LIN {X -0.093,Y -454.744,Z 848.526,A 0.000,B 0.000,C 90.000,E1 94.645} C_DIS
LIN {X 0.070,Y -444.193,Z 848.516,A 0.000,B 0.000,C 90.000,E1 92.808} C_DIS
LIN {X -0.166,Y -434.901,Z 848.507,A 0.000,B 0.000,C 90.000,E1 91.260} C_DIS
LIN {X -0.133,Y -425.303,Z 848.498,A 0.000,B 0.000,C 90.000,E1 89.656} C_DIS
LIN {X -0.064,Y -412.236,Z 848.486,A 0.000,B 0.000,C 90.000,E1 87.478} C_DIS
LIN {X 0.014,Y -402.403,Z 848.477,A 0.000,B 0.000,C 90.000,E1 85.812} C_DIS
LIN {X -0.027,Y -390.990,Z 848.466,A 0.000,B 0.000,C 90.000,E1 83.856} C_DIS
LIN {X 0.140,Y -378.162,Z 848.453,A 0.000,B 0.000,C 90.000,E1 81.546} C_DIS
LIN {X 0.095,Y -364.044,Z 848.439,A 0.000,B 0.000,C 90.000,E1 78.926} C_DIS
LIN {X -0.197,Y -351.890,Z 848.425,A 0.000,B 0.000,C 90.000,E1 76.589} C_DIS
LIN {X -0.106,Y -341.168,Z 848.414,A 0.000,B 0.000,C 90.000,E1 74.448} C_DIS
LIN {X 0.022,Y -327.690,Z 848.398,A 0.000,B 0.000,C 90.000,E1 71.638} C_DIS
LIN {X 0.142,Y -316.044,Z 848.384,A 0.000,B 0.000,C 90.000,E1 69.082} C_DIS
LIN {X -0.007,Y -301.999,Z 848.366,A 0.000,B 0.000,C 90.000,E1 65.869} C_DIS
LIN {X 0.053,Y -289.799,Z 848.349,A 0.000,B 0.000,C 90.000,E1 62.871} C_DIS
LIN {X -0.164,Y -279.159,Z 848.334,A 0.000,B 0.000,C 90.000,E1 60.205} C_DIS
LIN {X 0.005,Y -266.373,Z 848.315,A 0.000,B 0.000,C 90.000,E1 56.707} C_DIS
LIN {X 0.138,Y -254.533,Z 848.295,A 0.000,B 0.000,C 90.000,E1 53.130} C_DIS
LIN {X -0.031,Y -244.665,Z 848.277,A 0.000,B 0.000,C 90.000,E1 49.908} C_DIS
LIN {X -0.022,Y -234.511,Z 848.257,A 0.000,B 0.000,C 90.000,E1 46.215} C_DIS
LIN {X -0.016,Y -225.100,Z 848.236,A 0.000,B 0.000,C 90.000,E1 42.447} C_DIS
LIN {X 0.071,Y -218.003,Z 848.219,A 0.000,B 0.000,C 90.000,E1 39.358} C_DIS
LIN {X 0.029,Y -209.591,Z 848.197,A 0.000,B 0.000,C 90.000,E1 35.471} C_DIS
LIN {X -0.103,Y -203.336,Z 848.180,A 0.000,B 0.000,C 90.000,E1 32.339} C_DIS
LIN {X 0.075,Y -197.686,Z 848.162,A 0.000,B 0.000,C 90.000,E1 29.077} C_DIS
LIN {X 0.000,Y -192.660,Z 848.144,A 0.000,B 0.000,C 90.000,E1 25.848} C_DIS
LIN {X -0.094,Y -188.383,Z 848.125,A 0.000,B 0.000,C 90.000,E1 22.589} C_DIS
LIN {X -0.027,Y -184.224,Z 848.102,A 0.000,B 0.000,C 90.000,E1 18.417} C_DIS
LIN {X -0.080,Y -181.186,Z 848.079,A 0.000,B 0.000,C 90.000,E1 14.245} C_DIS
LIN {X -0.003,Y -178.587,Z 848.041,A 0.000,B 0.000,C 90.000,E1 7.466} C_DIS
LIN {X -0.048,Y -179.892,Z 847.979,A 0.000,B 0.000,C 90.000,E1 356.159} C_DIS
LIN {X -0.006,Y -182.801,Z 847.950,A 0.000,B 0.000,C 90.000,E1 351.084} C_DIS
LIN {X 0.036,Y -186.260,Z 847.927,A 0.000,B 0.000,C 90.000,E1 346.881} C_DIS
LIN {X 0.040,Y -190.786,Z 847.904,A 0.000,B 0.000,C 90.000,E1 342.725} C_DIS
LIN {X -0.070,Y -196.199,Z 847.881,A 0.000,B 0.000,C 90.000,E1 338.646} C_DIS
LIN {X -0.084,Y -202.510,Z 847.859,A 0.000,B 0.000,C 90.000,E1 334.588} C_DIS
LIN {X -0.101,Y -209.563,Z 847.836,A 0.000,B 0.000,C 90.000,E1 330.589} C_DIS
LIN {X -0.029,Y -217.357,Z 847.815,A 0.000,B 0.000,C 90.000,E1 326.628} C_DIS
LIN {X 0.070,Y -224.179,Z 847.797,A 0.000,B 0.000,C 90.000,E1 323.497} C_DIS
LIN {X 0.021,Y -232.765,Z 847.778,A 0.000,B 0.000,C 90.000,E1 320.070} C_DIS
LIN {X 0.005,Y -242.205,Z 847.759,A 0.000,B 0.000,C 90.000,E1 316.701} C_DIS
LIN {X 0.077,Y -252.624,Z 847.741,A 0.000,B 0.000,C 90.000,E1 313.380} C_DIS
LIN {X -0.055,Y -264.049,Z 847.723,A 0.000,B 0.000,C 90.000,E1 310.172} C_DIS
LIN {X 0.005,Y -276.404,Z 847.706,A 0.000,B 0.000,C 90.000,E1 306.996} C_DIS
LIN {X -0.026,Y -289.989,Z 847.688,A 0.000,B 0.000,C 90.000,E1 303.913} C_DIS
LIN {X -0.143,Y -304.691,Z 847.672,A 0.000,B 0.000,C 90.000,E1 300.924} C_DIS
LIN {X -0.023,Y -317.154,Z 847.659,A 0.000,B 0.000,C 90.000,E1 298.615} C_DIS
LIN {X 0.048,Y -332.889,Z 847.645,A 0.000,B 0.000,C 90.000,E1 296.052} C_DIS
LIN {X 0.102,Y -352.276,Z 847.629,A 0.000,B 0.000,C 90.000,E1 293.259} C_DIS
LIN {X 0.065,Y -371.074,Z 847.616,A 0.000,B 0.000,C 90.000,E1 290.865} C_DIS
LIN {X -0.046,Y -394.102,Z 847.602,A 0.000,B 0.000,C 90.000,E1 288.308} C_DIS
LIN {X -0.007,Y -412.240,Z 847.591,A 0.000,B 0.000,C 90.000,E1 286.386} C_DIS
LIN {X 0.017,Y -422.316,Z 847.585,A 0.000,B 0.000,C 90.000,E1 285.315} C_DIS
LIN {X -0.164,Y -434.613,Z 847.578,A 0.000,B 0.000,C 90.000,E1 284.008} C_DIS
LIN {X -0.130,Y -444.163,Z 847.572,A 0.000,B 0.000,C 90.000,E1 282.939} C_DIS
LIN {X -0.087,Y -453.154,Z 847.566,A 0.000,B 0.000,C 90.000,E1 281.883} C_DIS
LIN {X -0.023,Y -461.566,Z 847.560,A 0.000,B 0.000,C 90.000,E1 280.838} C_DIS
LIN {X 0.149,Y -469.405,Z 847.555,A 0.000,B 0.000,C 90.000,E1 279.792} C_DIS
LIN {X 0.168,Y -474.800,Z 847.550,A 0.000,B 0.000,C 90.000,E1 279.029} C_DIS
LIN {X 0.150,Y -479.624,Z 847.546,A 0.000,B 0.000,C 90.000,E1 278.276} C_DIS
LIN {X 0.114,Y -483.720,Z 847.542,A 0.000,B 0.000,C 90.000,E1 277.530} C_DIS
LIN {X 0.175,Y -487.070,Z 847.538,A 0.000,B 0.000,C 90.000,E1 276.777} C_DIS
LIN {X -0.110,Y -488.919,Z 847.535,A 0.000,B 0.000,C 90.000,E1 276.315} C_DIS
LIN {X 0.096,Y -490.405,Z 847.532,A 0.000,B 0.000,C 90.000,E1 275.796} C_DIS
LIN {X -0.176,Y -491.554,Z 847.530,A 0.000,B 0.000,C 90.000,E1 275.334} C_DIS
LIN {X 0.006,Y -492.300,Z 847.527,A 0.000,B 0.000,C 90.000,E1 274.821} C_DIS
LIN {X 0.238,Y -492.724,Z 847.524,A 0.000,B 0.000,C 90.000,E1 274.302} C_DIS
LIN {X -0.020,Y -492.771,Z 847.521,A 0.000,B 0.000,C 90.000,E1 273.841} C_DIS
LIN {X 0.185,Y -492.421,Z 847.519,A 0.000,B 0.000,C 90.000,E1 273.326} C_DIS
LIN {X -0.074,Y -491.691,Z 847.516,A 0.000,B 0.000,C 90.000,E1 272.865} C_DIS
LIN {X 0.131,Y -490.485,Z 847.513,A 0.000,B 0.000,C 90.000,E1 272.350} C_DIS
LIN {X -0.154,Y -488.845,Z 847.510,A 0.000,B 0.000,C 90.000,E1 271.892} C_DIS
LIN {X 0.057,Y -486.738,Z 847.508,A 0.000,B 0.000,C 90.000,E1 271.375} C_DIS
LIN {X 0.241,Y -483.997,Z 847.505,A 0.000,B 0.000,C 90.000,E1 270.859} C_DIS
LIN {X -0.074,Y -480.610,Z 847.502,A 0.000,B 0.000,C 90.000,E1 270.401} C_DIS
LIN {X -0.239,Y -478.699,Z 847.501,A 0.000,B 0.000,C 90.000,E1 270.172} C_DIS
LIN {X -0.100,Y -474.155,Z 847.498,A 0.000,B 0.000,C 90.000,E1 269.656} C_DIS
LIN {X 0.101,Y -468.795,Z 847.495,A 0.000,B 0.000,C 90.000,E1 269.141} C_DIS
LIN {X 0.136,Y -462.760,Z 847.493,A 0.000,B 0.000,C 90.000,E1 268.682} C_DIS
LIN {X -0.193,Y -459.346,Z 847.492,A 0.000,B 0.000,C 90.000,E1 268.511} C_DIS
LIN {X 0.175,Y -452.338,Z 847.490,A 0.000,B 0.000,C 90.000,E1 268.108} C_DIS
LIN {X 0.168,Y -445.005,Z 847.488,A 0.000,B 0.000,C 90.000,E1 267.822} C_DIS
LIN {X -0.214,Y -437.402,Z 847.487,A 0.000,B 0.000,C 90.000,E1 267.650} C_DIS
LIN {X -0.193,Y -428.427,Z 847.486,A 0.000,B 0.000,C 90.000,E1 267.478} C_DIS
LIN {X 0.039,Y -421.444,Z 847.485,A 0.000,B 0.000,C 90.000,E1 267.364} C_DIS
LIN {X 0.194,Y -415.603,Z 847.485,A 0.000,B 0.000,C 90.000,E1 267.306} C_DIS
LIN {X 0.058,Y -181.028,Z 847.485,A 0.000,B 0.000,C 90.000,E1 267.306} C_DIS
LIN {X 0.079,Y -180.786,Z 847.471,A 0.000,B 0.000,C 90.000,E1 264.723} C_DIS
LIN {X -0.027,Y -178.883,Z 847.443,A 0.000,B 0.000,C 90.000,E1 259.690} C_DIS
LIN {X 0.049,Y -175.926,Z 847.414,A 0.000,B 0.000,C 90.000,E1 254.574} C_DIS
LIN {X -0.005,Y -175.366,Z 847.410,A 0.000,B 0.000,C 90.000,E1 253.740} C_DIS
LIN {X 0.053,Y -172.144,Z 847.386,A 0.000,B 0.000,C 90.000,E1 249.444} C_DIS
LIN {X 0.030,Y -171.608,Z 847.381,A 0.000,B 0.000,C 90.000,E1 248.592} C_DIS
LIN {X 0.019,Y -167.831,Z 847.357,A 0.000,B 0.000,C 90.000,E1 244.280} C_DIS
LIN {X 0.036,Y -166.557,Z 847.347,A 0.000,B 0.000,C 90.000,E1 242.538} C_DIS
LIN {X -0.054,Y -162.551,Z 847.323,A 0.000,B 0.000,C 90.000,E1 238.201} C_DIS
LIN {X 0.006,Y -161.229,Z 847.313,A 0.000,B 0.000,C 90.000,E1 236.421} C_DIS
LIN {X 0.041,Y -157.235,Z 847.289,A 0.000,B 0.000,C 90.000,E1 231.984} C_DIS
LIN {X 0.064,Y -155.959,Z 847.279,A 0.000,B 0.000,C 90.000,E1 230.194} C_DIS
LIN {X 0.023,Y -152.213,Z 847.254,A 0.000,B 0.000,C 90.000,E1 225.729} C_DIS
LIN {X 0.043,Y -150.457,Z 847.239,A 0.000,B 0.000,C 90.000,E1 223.014} C_DIS
LIN {X 0.069,Y -147.183,Z 847.214,A 0.000,B 0.000,C 90.000,E1 218.463} C_DIS
LIN {X 0.036,Y -145.201,Z 847.194,A 0.000,B 0.000,C 90.000,E1 214.818} C_DIS
LIN {X -0.054,Y -142.338,Z 847.163,A 0.000,B 0.000,C 90.000,E1 209.333} C_DIS
LIN {X -0.001,Y -141.727,Z 847.153,A 0.000,B 0.000,C 90.000,E1 207.462} C_DIS
LIN {X -0.019,Y -139.480,Z 847.116,A 0.000,B 0.000,C 90.000,E1 200.972} C_DIS
LIN {X -0.029,Y -138.979,Z 847.101,A 0.000,B 0.000,C 90.000,E1 198.181} C_DIS
LIN {X -0.045,Y -138.332,Z 847.054,A 0.000,B 0.000,C 90.000,E1 189.782} C_DIS
LIN {X -0.044,Y -139.429,Z 847.008,A 0.000,B 0.000,C 90.000,E1 181.375} C_DIS
LIN {X 0.009,Y -141.357,Z 846.971,A 0.000,B 0.000,C 90.000,E1 174.837} C_DIS
LIN {X -0.015,Y -142.711,Z 846.956,A 0.000,B 0.000,C 90.000,E1 172.064} C_DIS
LIN {X -0.056,Y -145.085,Z 846.930,A 0.000,B 0.000,C 90.000,E1 167.465} C_DIS
LIN {X -0.061,Y -147.710,Z 846.910,A 0.000,B 0.000,C 90.000,E1 163.795} C_DIS
LIN {X 0.023,Y -150.365,Z 846.890,A 0.000,B 0.000,C 90.000,E1 160.115} C_DIS
LIN {X 0.041,Y -153.791,Z 846.869,A 0.000,B 0.000,C 90.000,E1 156.485} C_DIS
LIN {X -0.038,Y -157.204,Z 846.849,A 0.000,B 0.000,C 90.000,E1 152.922} C_DIS
LIN {X 0.043,Y -161.366,Z 846.830,A 0.000,B 0.000,C 90.000,E1 149.331} C_DIS
LIN {X 0.054,Y -165.568,Z 846.810,A 0.000,B 0.000,C 90.000,E1 145.801} C_DIS
LIN {X -0.062,Y -170.487,Z 846.791,A 0.000,B 0.000,C 90.000,E1 142.351} C_DIS
LIN {X 0.086,Y -175.367,Z 846.772,A 0.000,B 0.000,C 90.000,E1 138.852} C_DIS
LIN {X -0.051,Y -180.991,Z 846.753,A 0.000,B 0.000,C 90.000,E1 135.486} C_DIS
LIN {X 0.074,Y -186.419,Z 846.734,A 0.000,B 0.000,C 90.000,E1 132.081} C_DIS
LIN {X -0.125,Y -191.045,Z 846.720,A 0.000,B 0.000,C 90.000,E1 129.644} C_DIS
LIN {X -0.005,Y -192.945,Z 846.714,A 0.000,B 0.000,C 90.000,E1 128.463} C_DIS
LIN {X -0.055,Y -293.674,Z 846.714,A 0.000,B 0.000,C 90.000,E1 128.463} C_DIS
LIN {X -0.103,Y -294.466,Z 846.714,A 0.000,B 0.000,C 90.000,E1 128.463} C_DIS
LIN {X 0.120,Y -300.090,Z 846.712,A 0.000,B 0.000,C 90.000,E1 128.177} C_DIS
LIN {X -0.076,Y -302.819,Z 846.711,A 0.000,B 0.000,C 90.000,E1 127.971} C_DIS
LIN {X -0.016,Y -306.570,Z 846.708,A 0.000,B 0.000,C 90.000,E1 127.443} C_DIS
LIN {X -0.001,Y -308.236,Z 846.706,A 0.000,B 0.000,C 90.000,E1 127.111} C_DIS
LIN {X -0.044,Y -309.542,Z 846.704,A 0.000,B 0.000,C 90.000,E1 126.790} C_DIS
LIN {X 0.123,Y -321.746,Z 846.683,A 0.000,B 0.000,C 90.000,E1 122.880} C_DIS
LIN {X 0.002,Y -332.292,Z 846.667,A 0.000,B 0.000,C 90.000,E1 120.050} C_DIS
LIN {X -0.030,Y -344.201,Z 846.651,A 0.000,B 0.000,C 90.000,E1 117.257} C_DIS
LIN {X -0.025,Y -357.574,Z 846.636,A 0.000,B 0.000,C 90.000,E1 114.515} C_DIS
LIN {X -0.172,Y -370.791,Z 846.623,A 0.000,B 0.000,C 90.000,E1 112.153} C_DIS
LIN {X -0.133,Y -385.354,Z 846.610,A 0.000,B 0.000,C 90.000,E1 109.812} C_DIS
LIN {X 0.009,Y -401.370,Z 846.597,A 0.000,B 0.000,C 90.000,E1 107.511} C_DIS
LIN {X -0.078,Y -418.953,Z 846.585,A 0.000,B 0.000,C 90.000,E1 105.300} C_DIS
LIN {X 0.079,Y -438.195,Z 846.573,A 0.000,B 0.000,C 90.000,E1 103.119} C_DIS
LIN {X -0.120,Y -458.364,Z 846.562,A 0.000,B 0.000,C 90.000,E1 101.130} C_DIS
LIN {X -0.212,Y -468.460,Z 846.557,A 0.000,B 0.000,C 90.000,E1 100.197} C_DIS
LIN {X -0.174,Y -470.265,Z 846.555,A 0.000,B 0.000,C 90.000,E1 99.962} C_DIS
LIN {X 0.141,Y -471.770,Z 846.554,A 0.000,B 0.000,C 90.000,E1 99.670} C_DIS
LIN {X -0.087,Y -472.896,Z 846.552,A 0.000,B 0.000,C 90.000,E1 99.443} C_DIS
LIN {X 0.097,Y -474.241,Z 846.550,A 0.000,B 0.000,C 90.000,E1 98.916} C_DIS
LIN {X 0.214,Y -474.566,Z 846.547,A 0.000,B 0.000,C 90.000,E1 98.398} C_DIS
LIN {X -0.128,Y -473.929,Z 846.544,A 0.000,B 0.000,C 90.000,E1 97.936} C_DIS
LIN {X 0.063,Y -472.229,Z 846.541,A 0.000,B 0.000,C 90.000,E1 97.409} C_DIS
LIN {X -0.138,Y -470.887,Z 846.540,A 0.000,B 0.000,C 90.000,E1 97.182} C_DIS
LIN {X -0.206,Y -454.710,Z 846.526,A 0.000,B 0.000,C 90.000,E1 94.645} C_DIS
LIN {X -0.041,Y -444.143,Z 846.516,A 0.000,B 0.000,C 90.000,E1 92.808} C_DIS
LIN {X 0.159,Y -434.848,Z 846.507,A 0.000,B 0.000,C 90.000,E1 91.203} C_DIS
LIN {X 0.184,Y -425.251,Z 846.498,A 0.000,B 0.000,C 90.000,E1 89.599} C_DIS
LIN {X -0.171,Y -412.180,Z 846.486,A 0.000,B 0.000,C 90.000,E1 87.478} C_DIS
LIN {X -0.090,Y -402.341,Z 846.477,A 0.000,B 0.000,C 90.000,E1 85.812} C_DIS
LIN {X -0.131,Y -390.926,Z 846.466,A 0.000,B 0.000,C 90.000,E1 83.856} C_DIS
LIN {X 0.040,Y -378.086,Z 846.453,A 0.000,B 0.000,C 90.000,E1 81.546} C_DIS
LIN {X -0.003,Y -363.983,Z 846.438,A 0.000,B 0.000,C 90.000,E1 78.926} C_DIS
LIN {X 0.047,Y -351.842,Z 846.425,A 0.000,B 0.000,C 90.000,E1 76.533} C_DIS
LIN {X 0.128,Y -341.179,Z 846.413,A 0.000,B 0.000,C 90.000,E1 74.393} C_DIS
LIN {X -0.069,Y -327.733,Z 846.398,A 0.000,B 0.000,C 90.000,E1 71.638} C_DIS
LIN {X 0.056,Y -316.089,Z 846.384,A 0.000,B 0.000,C 90.000,E1 69.082} C_DIS
LIN {X 0.036,Y -302.071,Z 846.366,A 0.000,B 0.000,C 90.000,E1 65.845} C_DIS
LIN {X -0.023,Y -289.895,Z 846.349,A 0.000,B 0.000,C 90.000,E1 62.871} C_DIS
LIN {X 0.148,Y -279.335,Z 846.334,A 0.000,B 0.000,C 90.000,E1 60.127} C_DIS
LIN {X -0.055,Y -266.613,Z 846.315,A 0.000,B 0.000,C 90.000,E1 56.707} C_DIS
LIN {X 0.053,Y -255.972,Z 846.297,A 0.000,B 0.000,C 90.000,E1 53.497} C_DIS
LIN {X -0.070,Y -244.986,Z 846.277,A 0.000,B 0.000,C 90.000,E1 49.908} C_DIS
LIN {X -0.050,Y -234.827,Z 846.257,A 0.000,B 0.000,C 90.000,E1 46.215} C_DIS
LIN {X -0.034,Y -225.429,Z 846.236,A 0.000,B 0.000,C 90.000,E1 42.447} C_DIS
LIN {X 0.062,Y -218.321,Z 846.219,A 0.000,B 0.000,C 90.000,E1 39.358} C_DIS
LIN {X 0.030,Y -209.918,Z 846.197,A 0.000,B 0.000,C 90.000,E1 35.471} C_DIS
LIN {X 0.003,Y -202.175,Z 846.175,A 0.000,B 0.000,C 90.000,E1 31.514} C_DIS
LIN {X 0.046,Y -196.669,Z 846.157,A 0.000,B 0.000,C 90.000,E1 28.281} C_DIS
LIN {X 0.031,Y -191.823,Z 846.139,A 0.000,B 0.000,C 90.000,E1 25.027} C_DIS
LIN {X 0.089,Y -187.751,Z 846.121,A 0.000,B 0.000,C 90.000,E1 21.716} C_DIS
LIN {X 0.010,Y -183.833,Z 846.098,A 0.000,B 0.000,C 90.000,E1 17.583} C_DIS
LIN {X 0.053,Y -180.603,Z 846.070,A 0.000,B 0.000,C 90.000,E1 12.535} C_DIS
LIN {X 0.030,Y -178.550,Z 846.027,A 0.000,B 0.000,C 90.000,E1 4.935} C_DIS
LIN {X -0.040,Y -180.220,Z 845.979,A 0.000,B 0.000,C 90.000,E1 356.159} C_DIS
LIN {X 0.014,Y -183.148,Z 845.951,A 0.000,B 0.000,C 90.000,E1 351.084} C_DIS
LIN {X 0.067,Y -186.608,Z 845.927,A 0.000,B 0.000,C 90.000,E1 346.881} C_DIS
LIN {X 0.083,Y -191.114,Z 845.904,A 0.000,B 0.000,C 90.000,E1 342.725} C_DIS
LIN {X -0.017,Y -196.494,Z 845.881,A 0.000,B 0.000,C 90.000,E1 338.646} C_DIS
LIN {X -0.019,Y -202.772,Z 845.859,A 0.000,B 0.000,C 90.000,E1 334.588} C_DIS
LIN {X -0.026,Y -209.784,Z 845.837,A 0.000,B 0.000,C 90.000,E1 330.589} C_DIS
LIN {X 0.056,Y -217.581,Z 845.815,A 0.000,B 0.000,C 90.000,E1 326.628} C_DIS
LIN {X -0.016,Y -224.409,Z 845.797,A 0.000,B 0.000,C 90.000,E1 323.543} C_DIS
LIN {X -0.053,Y -232.977,Z 845.778,A 0.000,B 0.000,C 90.000,E1 320.114} C_DIS
LIN {X -0.057,Y -242.395,Z 845.760,A 0.000,B 0.000,C 90.000,E1 316.743} C_DIS
LIN {X 0.029,Y -252.789,Z 845.741,A 0.000,B 0.000,C 90.000,E1 313.419} C_DIS
LIN {X 0.079,Y -264.179,Z 845.723,A 0.000,B 0.000,C 90.000,E1 310.172} C_DIS
LIN {X -0.017,Y -276.475,Z 845.706,A 0.000,B 0.000,C 90.000,E1 307.030} C_DIS
LIN {X 0.128,Y -289.994,Z 845.689,A 0.000,B 0.000,C 90.000,E1 303.913} C_DIS
LIN {X 0.017,Y -304.644,Z 845.672,A 0.000,B 0.000,C 90.000,E1 300.924} C_DIS
LIN {X 0.143,Y -317.065,Z 845.659,A 0.000,B 0.000,C 90.000,E1 298.615} C_DIS
LIN {X -0.080,Y -332.737,Z 845.645,A 0.000,B 0.000,C 90.000,E1 296.104} C_DIS
LIN {X -0.024,Y -354.247,Z 845.628,A 0.000,B 0.000,C 90.000,E1 293.003} C_DIS
LIN {X -0.104,Y -370.737,Z 845.616,A 0.000,B 0.000,C 90.000,E1 290.918} C_DIS
LIN {X -0.082,Y -393.490,Z 845.602,A 0.000,B 0.000,C 90.000,E1 288.362} C_DIS
LIN {X -0.044,Y -411.553,Z 845.591,A 0.000,B 0.000,C 90.000,E1 286.441} C_DIS
LIN {X -0.048,Y -421.673,Z 845.585,A 0.000,B 0.000,C 90.000,E1 285.371} C_DIS
LIN {X -0.197,Y -433.922,Z 845.578,A 0.000,B 0.000,C 90.000,E1 284.064} C_DIS
LIN {X 0.160,Y -443.513,Z 845.572,A 0.000,B 0.000,C 90.000,E1 282.952} C_DIS
LIN {X -0.233,Y -452.565,Z 845.566,A 0.000,B 0.000,C 90.000,E1 281.951} C_DIS
LIN {X -0.086,Y -461.010,Z 845.560,A 0.000,B 0.000,C 90.000,E1 280.894} C_DIS
LIN {X 0.076,Y -468.915,Z 845.555,A 0.000,B 0.000,C 90.000,E1 279.849} C_DIS
LIN {X 0.015,Y -474.349,Z 845.551,A 0.000,B 0.000,C 90.000,E1 279.095} C_DIS
LIN {X -0.004,Y -479.246,Z 845.546,A 0.000,B 0.000,C 90.000,E1 278.341} C_DIS
LIN {X 0.024,Y -483.378,Z 845.542,A 0.000,B 0.000,C 90.000,E1 277.587} C_DIS
LIN {X 0.082,Y -486.790,Z 845.538,A 0.000,B 0.000,C 90.000,E1 276.834} C_DIS
LIN {X -0.206,Y -488.674,Z 845.535,A 0.000,B 0.000,C 90.000,E1 276.372} C_DIS
LIN {X -0.003,Y -490.202,Z 845.533,A 0.000,B 0.000,C 90.000,E1 275.853} C_DIS
LIN {X 0.212,Y -491.416,Z 845.530,A 0.000,B 0.000,C 90.000,E1 275.334} C_DIS
LIN {X -0.097,Y -492.197,Z 845.527,A 0.000,B 0.000,C 90.000,E1 274.878} C_DIS
LIN {X 0.135,Y -492.667,Z 845.524,A 0.000,B 0.000,C 90.000,E1 274.359} C_DIS
LIN {X -0.124,Y -492.759,Z 845.522,A 0.000,B 0.000,C 90.000,E1 273.898} C_DIS
LIN {X 0.079,Y -492.465,Z 845.519,A 0.000,B 0.000,C 90.000,E1 273.383} C_DIS
LIN {X -0.179,Y -491.794,Z 845.516,A 0.000,B 0.000,C 90.000,E1 272.922} C_DIS
LIN {X 0.026,Y -490.669,Z 845.513,A 0.000,B 0.000,C 90.000,E1 272.407} C_DIS
LIN {X 0.230,Y -489.120,Z 845.511,A 0.000,B 0.000,C 90.000,E1 271.892} C_DIS
LIN {X -0.047,Y -487.059,Z 845.508,A 0.000,B 0.000,C 90.000,E1 271.432} C_DIS
LIN {X 0.141,Y -484.453,Z 845.505,A 0.000,B 0.000,C 90.000,E1 270.917} C_DIS
LIN {X -0.173,Y -481.145,Z 845.502,A 0.000,B 0.000,C 90.000,E1 270.458} C_DIS
LIN {X -0.020,Y -477.198,Z 845.500,A 0.000,B 0.000,C 90.000,E1 269.943} C_DIS
LIN {X 0.110,Y -472.290,Z 845.497,A 0.000,B 0.000,C 90.000,E1 269.427} C_DIS
LIN {X 0.005,Y -469.665,Z 845.496,A 0.000,B 0.000,C 90.000,E1 269.198} C_DIS
LIN {X -0.005,Y -463.797,Z 845.493,A 0.000,B 0.000,C 90.000,E1 268.740} C_DIS
LIN {X 0.087,Y -460.414,Z 845.492,A 0.000,B 0.000,C 90.000,E1 268.511} C_DIS
LIN {X -0.074,Y -453.517,Z 845.490,A 0.000,B 0.000,C 90.000,E1 268.165} C_DIS
LIN {X -0.170,Y -446.226,Z 845.488,A 0.000,B 0.000,C 90.000,E1 267.879} C_DIS
LIN {X -0.190,Y -438.569,Z 845.487,A 0.000,B 0.000,C 90.000,E1 267.650} C_DIS
LIN {X -0.206,Y -430.047,Z 845.486,A 0.000,B 0.000,C 90.000,E1 267.478} C_DIS
LIN {X 0.199,Y -420.197,Z 845.485,A 0.000,B 0.000,C 90.000,E1 267.306} C_DIS
LIN {X 0.055,Y -416.039,Z 845.485,A 0.000,B 0.000,C 90.000,E1 267.306} C_DIS
LIN {X -0.007,Y -181.025,Z 845.485,A 0.000,B 0.000,C 90.000,E1 267.306} C_DIS
LIN {X 0.014,Y -180.778,Z 845.471,A 0.000,B 0.000,C 90.000,E1 264.723} C_DIS
LIN {X -0.091,Y -178.874,Z 845.443,A 0.000,B 0.000,C 90.000,E1 259.690} C_DIS
LIN {X -0.015,Y -175.917,Z 845.414,A 0.000,B 0.000,C 90.000,E1 254.574} C_DIS
LIN {X 0.041,Y -174.611,Z 845.405,A 0.000,B 0.000,C 90.000,E1 252.851} C_DIS
LIN {X -0.033,Y -171.592,Z 845.381,A 0.000,B 0.000,C 90.000,E1 248.592} C_DIS
LIN {X -0.044,Y -167.814,Z 845.357,A 0.000,B 0.000,C 90.000,E1 244.280} C_DIS
LIN {X -0.026,Y -166.536,Z 845.347,A 0.000,B 0.000,C 90.000,E1 242.538} C_DIS
LIN {X 0.024,Y -162.534,Z 845.323,A 0.000,B 0.000,C 90.000,E1 238.152} C_DIS
LIN {X -0.055,Y -161.210,Z 845.313,A 0.000,B 0.000,C 90.000,E1 236.421} C_DIS
LIN {X -0.019,Y -157.219,Z 845.289,A 0.000,B 0.000,C 90.000,E1 231.984} C_DIS
LIN {X 0.004,Y -155.945,Z 845.279,A 0.000,B 0.000,C 90.000,E1 230.194} C_DIS
LIN {X -0.036,Y -152.198,Z 845.254,A 0.000,B 0.000,C 90.000,E1 225.729} C_DIS
LIN {X -0.015,Y -150.444,Z 845.239,A 0.000,B 0.000,C 90.000,E1 223.014} C_DIS
LIN {X 0.012,Y -147.170,Z 845.214,A 0.000,B 0.000,C 90.000,E1 218.463} C_DIS
LIN {X -0.022,Y -145.186,Z 845.193,A 0.000,B 0.000,C 90.000,E1 214.818} C_DIS
LIN {X 0.014,Y -142.330,Z 845.163,A 0.000,B 0.000,C 90.000,E1 209.283} C_DIS
LIN {X -0.057,Y -141.718,Z 845.152,A 0.000,B 0.000,C 90.000,E1 207.462} C_DIS
LIN {X 0.056,Y -139.476,Z 845.116,A 0.000,B 0.000,C 90.000,E1 200.918} C_DIS
LIN {X 0.047,Y -138.973,Z 845.101,A 0.000,B 0.000,C 90.000,E1 198.127} C_DIS
LIN {X 0.037,Y -138.330,Z 845.054,A 0.000,B 0.000,C 90.000,E1 189.726} C_DIS
LIN {X 0.039,Y -139.435,Z 845.007,A 0.000,B 0.000,C 90.000,E1 181.318} C_DIS
LIN {X -0.021,Y -140.963,Z 844.976,A 0.000,B 0.000,C 90.000,E1 175.755} C_DIS
LIN {X 0.070,Y -142.719,Z 844.956,A 0.000,B 0.000,C 90.000,E1 172.008} C_DIS
LIN {X 0.029,Y -145.099,Z 844.930,A 0.000,B 0.000,C 90.000,E1 167.409} C_DIS
LIN {X 0.023,Y -147.723,Z 844.910,A 0.000,B 0.000,C 90.000,E1 163.740} C_DIS
LIN {X -0.035,Y -150.383,Z 844.889,A 0.000,B 0.000,C 90.000,E1 160.115} C_DIS
LIN {X -0.018,Y -153.815,Z 844.869,A 0.000,B 0.000,C 90.000,E1 156.485} C_DIS
LIN {X 0.042,Y -157.226,Z 844.849,A 0.000,B 0.000,C 90.000,E1 152.871} C_DIS
LIN {X -0.018,Y -161.394,Z 844.830,A 0.000,B 0.000,C 90.000,E1 149.331} C_DIS
LIN {X -0.008,Y -165.596,Z 844.810,A 0.000,B 0.000,C 90.000,E1 145.801} C_DIS
LIN {X -0.021,Y -170.519,Z 844.791,A 0.000,B 0.000,C 90.000,E1 142.316} C_DIS
LIN {X 0.023,Y -175.399,Z 844.771,A 0.000,B 0.000,C 90.000,E1 138.852} C_DIS
LIN {X 0.013,Y -181.023,Z 844.753,A 0.000,B 0.000,C 90.000,E1 135.445} C_DIS
LIN {X 0.007,Y -186.454,Z 844.734,A 0.000,B 0.000,C 90.000,E1 132.081} C_DIS
LIN {X 0.077,Y -191.078,Z 844.720,A 0.000,B 0.000,C 90.000,E1 129.564} C_DIS
LIN {X 0.014,Y -192.935,Z 844.714,A 0.000,B 0.000,C 90.000,E1 128.463} C_DIS
LIN {X -0.015,Y -293.729,Z 844.714,A 0.000,B 0.000,C 90.000,E1 128.463} C_DIS
LIN {X 0.026,Y -295.732,Z 844.713,A 0.000,B 0.000,C 90.000,E1 128.418} C_DIS
LIN {X 0.016,Y -300.426,Z 844.712,A 0.000,B 0.000,C 90.000,E1 128.177} C_DIS
LIN {X 0.005,Y -303.037,Z 844.711,A 0.000,B 0.000,C 90.000,E1 127.935} C_DIS
LIN {X 0.017,Y -306.793,Z 844.708,A 0.000,B 0.000,C 90.000,E1 127.397} C_DIS
LIN {X -0.025,Y -308.400,Z 844.706,A 0.000,B 0.000,C 90.000,E1 127.076} C_DIS
LIN {X -0.007,Y -309.661,Z 844.704,A 0.000,B 0.000,C 90.000,E1 126.744} C_DIS
LIN {X 0.100,Y -320.761,Z 844.684,A 0.000,B 0.000,C 90.000,E1 123.166} C_DIS
LIN {X -0.045,Y -331.180,Z 844.668,A 0.000,B 0.000,C 90.000,E1 120.335} C_DIS
LIN {X 0.062,Y -342.949,Z 844.653,A 0.000,B 0.000,C 90.000,E1 117.513} C_DIS
LIN {X 0.030,Y -356.178,Z 844.638,A 0.000,B 0.000,C 90.000,E1 114.771} C_DIS
LIN {X -0.007,Y -369.252,Z 844.624,A 0.000,B 0.000,C 90.000,E1 112.386} C_DIS
LIN {X -0.139,Y -383.663,Z 844.611,A 0.000,B 0.000,C 90.000,E1 110.066} C_DIS
LIN {X -0.032,Y -399.514,Z 844.599,A 0.000,B 0.000,C 90.000,E1 107.764} C_DIS
LIN {X -0.156,Y -416.919,Z 844.586,A 0.000,B 0.000,C 90.000,E1 105.552} C_DIS
LIN {X 0.036,Y -436.001,Z 844.574,A 0.000,B 0.000,C 90.000,E1 103.355} C_DIS
LIN {X 0.222,Y -456.106,Z 844.563,A 0.000,B 0.000,C 90.000,E1 101.299} C_DIS
LIN {X 0.061,Y -466.368,Z 844.558,A 0.000,B 0.000,C 90.000,E1 100.366} C_DIS
LIN {X 0.019,Y -468.688,Z 844.556,A 0.000,B 0.000,C 90.000,E1 100.141} C_DIS
LIN {X 0.060,Y -470.443,Z 844.555,A 0.000,B 0.000,C 90.000,E1 99.905} C_DIS
LIN {X -0.088,Y -471.910,Z 844.554,A 0.000,B 0.000,C 90.000,E1 99.670} C_DIS
LIN {X 0.228,Y -473.004,Z 844.552,A 0.000,B 0.000,C 90.000,E1 99.378} C_DIS
LIN {X -0.132,Y -474.298,Z 844.549,A 0.000,B 0.000,C 90.000,E1 98.916} C_DIS
LIN {X -0.013,Y -474.580,Z 844.547,A 0.000,B 0.000,C 90.000,E1 98.398} C_DIS
LIN {X 0.179,Y -473.898,Z 844.544,A 0.000,B 0.000,C 90.000,E1 97.871} C_DIS
LIN {X -0.163,Y -472.144,Z 844.541,A 0.000,B 0.000,C 90.000,E1 97.409} C_DIS
LIN {X 0.103,Y -470.766,Z 844.540,A 0.000,B 0.000,C 90.000,E1 97.125} C_DIS
LIN {X 0.026,Y -454.591,Z 844.526,A 0.000,B 0.000,C 90.000,E1 94.588} C_DIS
LIN {X 0.184,Y -444.029,Z 844.515,A 0.000,B 0.000,C 90.000,E1 92.751} C_DIS
LIN {X -0.057,Y -434.716,Z 844.507,A 0.000,B 0.000,C 90.000,E1 91.203} C_DIS
LIN {X -0.029,Y -425.116,Z 844.498,A 0.000,B 0.000,C 90.000,E1 89.599} C_DIS
LIN {X 0.031,Y -412.038,Z 844.486,A 0.000,B 0.000,C 90.000,E1 87.421} C_DIS
LIN {X 0.104,Y -402.189,Z 844.477,A 0.000,B 0.000,C 90.000,E1 85.755} C_DIS
LIN {X 0.053,Y -390.776,Z 844.466,A 0.000,B 0.000,C 90.000,E1 83.799} C_DIS
LIN {X -0.184,Y -379.522,Z 844.455,A 0.000,B 0.000,C 90.000,E1 81.837} C_DIS
LIN {X 0.171,Y -365.390,Z 844.440,A 0.000,B 0.000,C 90.000,E1 79.162} C_DIS
LIN {X -0.066,Y -351.733,Z 844.425,A 0.000,B 0.000,C 90.000,E1 76.520} C_DIS
LIN {X -0.063,Y -341.109,Z 844.413,A 0.000,B 0.000,C 90.000,E1 74.393} C_DIS
LIN {X 0.056,Y -327.694,Z 844.398,A 0.000,B 0.000,C 90.000,E1 71.583} C_DIS
LIN {X -0.124,Y -316.063,Z 844.384,A 0.000,B 0.000,C 90.000,E1 69.082} C_DIS
LIN {X 0.139,Y -302.072,Z 844.366,A 0.000,B 0.000,C 90.000,E1 65.793} C_DIS
LIN {X 0.070,Y -289.923,Z 844.349,A 0.000,B 0.000,C 90.000,E1 62.820} C_DIS
LIN {X -0.010,Y -279.443,Z 844.334,A 0.000,B 0.000,C 90.000,E1 60.127} C_DIS
LIN {X 0.168,Y -266.798,Z 844.315,A 0.000,B 0.000,C 90.000,E1 56.628} C_DIS
LIN {X -0.082,Y -256.218,Z 844.297,A 0.000,B 0.000,C 90.000,E1 53.497} C_DIS
LIN {X -0.005,Y -245.256,Z 844.277,A 0.000,B 0.000,C 90.000,E1 49.865} C_DIS
LIN {X 0.003,Y -235.088,Z 844.257,A 0.000,B 0.000,C 90.000,E1 46.176} C_DIS
LIN {X 0.037,Y -225.721,Z 844.236,A 0.000,B 0.000,C 90.000,E1 42.405} C_DIS
LIN {X -0.025,Y -218.594,Z 844.219,A 0.000,B 0.000,C 90.000,E1 39.358} C_DIS
LIN {X 0.077,Y -210.204,Z 844.197,A 0.000,B 0.000,C 90.000,E1 35.438} C_DIS
LIN {X 0.012,Y -203.937,Z 844.179,A 0.000,B 0.000,C 90.000,E1 32.291} C_DIS
LIN {X 0.035,Y -198.265,Z 844.162,A 0.000,B 0.000,C 90.000,E1 29.077} C_DIS
LIN {X -0.025,Y -193.254,Z 844.144,A 0.000,B 0.000,C 90.000,E1 25.848} C_DIS
LIN {X -0.105,Y -188.990,Z 844.125,A 0.000,B 0.000,C 90.000,E1 22.589} C_DIS
LIN {X -0.018,Y -184.803,Z 844.102,A 0.000,B 0.000,C 90.000,E1 18.417} C_DIS
LIN {X -0.075,Y -181.342,Z 844.074,A 0.000,B 0.000,C 90.000,E1 13.411} C_DIS
LIN {X -0.081,Y -179.062,Z 844.037,A 0.000,B 0.000,C 90.000,E1 6.663} C_DIS
LIN {X -0.033,Y -180.539,Z 843.979,A 0.000,B 0.000,C 90.000,E1 356.159} C_DIS
LIN {X 0.034,Y -183.499,Z 843.951,A 0.000,B 0.000,C 90.000,E1 351.084} C_DIS
LIN {X -0.084,Y -186.956,Z 843.927,A 0.000,B 0.000,C 90.000,E1 346.937} C_DIS
LIN {X -0.058,Y -191.438,Z 843.904,A 0.000,B 0.000,C 90.000,E1 342.779} C_DIS
LIN {X 0.037,Y -196.782,Z 843.881,A 0.000,B 0.000,C 90.000,E1 338.646} C_DIS
LIN {X 0.045,Y -203.022,Z 843.859,A 0.000,B 0.000,C 90.000,E1 334.588} C_DIS
LIN {X 0.048,Y -210.013,Z 843.837,A 0.000,B 0.000,C 90.000,E1 330.589} C_DIS
LIN {X 0.140,Y -217.801,Z 843.815,A 0.000,B 0.000,C 90.000,E1 326.628} C_DIS
LIN {X -0.057,Y -224.639,Z 843.798,A 0.000,B 0.000,C 90.000,E1 323.577} C_DIS
LIN {X 0.049,Y -233.185,Z 843.779,A 0.000,B 0.000,C 90.000,E1 320.114} C_DIS
LIN {X 0.055,Y -242.574,Z 843.760,A 0.000,B 0.000,C 90.000,E1 316.743} C_DIS
LIN {X -0.032,Y -252.954,Z 843.741,A 0.000,B 0.000,C 90.000,E1 313.461} C_DIS
LIN {X 0.010,Y -264.299,Z 843.723,A 0.000,B 0.000,C 90.000,E1 310.216} C_DIS
LIN {X -0.097,Y -276.552,Z 843.706,A 0.000,B 0.000,C 90.000,E1 307.076} C_DIS
LIN {X -0.124,Y -289.998,Z 843.689,A 0.000,B 0.000,C 90.000,E1 303.992} C_DIS
LIN {X 0.175,Y -304.587,Z 843.672,A 0.000,B 0.000,C 90.000,E1 300.924} C_DIS
LIN {X -0.124,Y -316.970,Z 843.659,A 0.000,B 0.000,C 90.000,E1 298.693} C_DIS
LIN {X 0.089,Y -332.579,Z 843.645,A 0.000,B 0.000,C 90.000,E1 296.104} C_DIS
LIN {X -0.013,Y -351.734,Z 843.630,A 0.000,B 0.000,C 90.000,E1 293.334} C_DIS
LIN {X 0.070,Y -370.404,Z 843.616,A 0.000,B 0.000,C 90.000,E1 290.918} C_DIS
LIN {X 0.207,Y -395.786,Z 843.600,A 0.000,B 0.000,C 90.000,E1 288.055} C_DIS
LIN {X 0.056,Y -411.195,Z 843.591,A 0.000,B 0.000,C 90.000,E1 286.441} C_DIS
LIN {X 0.078,Y -421.294,Z 843.585,A 0.000,B 0.000,C 90.000,E1 285.371} C_DIS
LIN {X -0.061,Y -433.545,Z 843.578,A 0.000,B 0.000,C 90.000,E1 284.064} C_DIS
LIN {X -0.138,Y -443.142,Z 843.572,A 0.000,B 0.000,C 90.000,E1 283.008} C_DIS
LIN {X -0.101,Y -452.243,Z 843.566,A 0.000,B 0.000,C 90.000,E1 281.951} C_DIS
LIN {X 0.044,Y -460.709,Z 843.561,A 0.000,B 0.000,C 90.000,E1 280.894} C_DIS
LIN {X 0.206,Y -468.651,Z 843.555,A 0.000,B 0.000,C 90.000,E1 279.849} C_DIS
LIN {X 0.143,Y -474.126,Z 843.551,A 0.000,B 0.000,C 90.000,E1 279.095} C_DIS
LIN {X 0.124,Y -479.025,Z 843.546,A 0.000,B 0.000,C 90.000,E1 278.341} C_DIS
LIN {X -0.138,Y -481.879,Z 843.544,A 0.000,B 0.000,C 90.000,E1 277.871} C_DIS
LIN {X -0.154,Y -485.553,Z 843.539,A 0.000,B 0.000,C 90.000,E1 277.125} C_DIS
LIN {X -0.079,Y -488.519,Z 843.535,A 0.000,B 0.000,C 90.000,E1 276.372} C_DIS
LIN {X 0.124,Y -490.077,Z 843.533,A 0.000,B 0.000,C 90.000,E1 275.853} C_DIS
LIN {X -0.151,Y -491.279,Z 843.530,A 0.000,B 0.000,C 90.000,E1 275.391} C_DIS
LIN {X 0.027,Y -492.129,Z 843.527,A 0.000,B 0.000,C 90.000,E1 274.878} C_DIS
LIN {X -0.232,Y -492.644,Z 843.524,A 0.000,B 0.000,C 90.000,E1 274.416} C_DIS
LIN {X 0.000,Y -492.718,Z 843.522,A 0.000,B 0.000,C 90.000,E1 273.898} C_DIS
LIN {X 0.203,Y -492.452,Z 843.519,A 0.000,B 0.000,C 90.000,E1 273.383} C_DIS
LIN {X -0.056,Y -491.837,Z 843.516,A 0.000,B 0.000,C 90.000,E1 272.922} C_DIS
LIN {X 0.149,Y -490.756,Z 843.513,A 0.000,B 0.000,C 90.000,E1 272.407} C_DIS
LIN {X -0.136,Y -489.235,Z 843.511,A 0.000,B 0.000,C 90.000,E1 271.949} C_DIS
LIN {X 0.076,Y -487.234,Z 843.508,A 0.000,B 0.000,C 90.000,E1 271.432} C_DIS
LIN {X -0.221,Y -484.656,Z 843.505,A 0.000,B 0.000,C 90.000,E1 270.974} C_DIS
LIN {X -0.050,Y -481.446,Z 843.503,A 0.000,B 0.000,C 90.000,E1 270.458} C_DIS
LIN {X 0.103,Y -477.565,Z 843.500,A 0.000,B 0.000,C 90.000,E1 269.943} C_DIS
LIN {X 0.233,Y -472.749,Z 843.497,A 0.000,B 0.000,C 90.000,E1 269.427} C_DIS
LIN {X 0.102,Y -470.142,Z 843.496,A 0.000,B 0.000,C 90.000,E1 269.198} C_DIS
LIN {X 0.049,Y -464.243,Z 843.493,A 0.000,B 0.000,C 90.000,E1 268.740} C_DIS
LIN {X 0.124,Y -460.928,Z 843.492,A 0.000,B 0.000,C 90.000,E1 268.511} C_DIS
LIN {X -0.103,Y -454.106,Z 843.490,A 0.000,B 0.000,C 90.000,E1 268.165} C_DIS
LIN {X 0.175,Y -446.701,Z 843.488,A 0.000,B 0.000,C 90.000,E1 267.822} C_DIS
LIN {X 0.101,Y -438.850,Z 843.487,A 0.000,B 0.000,C 90.000,E1 267.593} C_DIS
LIN {X 0.078,Y -430.388,Z 843.486,A 0.000,B 0.000,C 90.000,E1 267.421} C_DIS
LIN {X 0.036,Y -420.265,Z 843.485,A 0.000,B 0.000,C 90.000,E1 267.306} C_DIS
LIN {X -0.104,Y -415.828,Z 843.485,A 0.000,B 0.000,C 90.000,E1 267.306} C_DIS
LIN {X -0.076,Y -181.023,Z 843.485,A 0.000,B 0.000,C 90.000,E1 267.306} C_DIS
LIN {X -0.053,Y -180.770,Z 843.471,A 0.000,B 0.000,C 90.000,E1 264.723} C_DIS
LIN {X 0.018,Y -178.864,Z 843.442,A 0.000,B 0.000,C 90.000,E1 259.634} C_DIS
LIN {X -0.081,Y -175.908,Z 843.414,A 0.000,B 0.000,C 90.000,E1 254.574} C_DIS
LIN {X 0.027,Y -174.592,Z 843.405,A 0.000,B 0.000,C 90.000,E1 252.834} C_DIS
LIN {X 0.062,Y -171.575,Z 843.381,A 0.000,B 0.000,C 90.000,E1 248.539} C_DIS
LIN {X 0.043,Y -167.799,Z 843.357,A 0.000,B 0.000,C 90.000,E1 244.229} C_DIS
LIN {X 0.058,Y -166.516,Z 843.347,A 0.000,B 0.000,C 90.000,E1 242.487} C_DIS
LIN {X 0.054,Y -163.224,Z 843.328,A 0.000,B 0.000,C 90.000,E1 238.997} C_DIS
LIN {X 0.017,Y -161.190,Z 843.313,A 0.000,B 0.000,C 90.000,E1 236.373} C_DIS
LIN {X -0.081,Y -157.201,Z 843.289,A 0.000,B 0.000,C 90.000,E1 231.984} C_DIS
LIN {X -0.057,Y -155.929,Z 843.279,A 0.000,B 0.000,C 90.000,E1 230.194} C_DIS
LIN {X 0.012,Y -152.181,Z 843.254,A 0.000,B 0.000,C 90.000,E1 225.688} C_DIS
LIN {X 0.028,Y -150.428,Z 843.239,A 0.000,B 0.000,C 90.000,E1 222.975} C_DIS
LIN {X -0.047,Y -147.156,Z 843.214,A 0.000,B 0.000,C 90.000,E1 218.463} C_DIS
LIN {X -0.079,Y -145.170,Z 843.193,A 0.000,B 0.000,C 90.000,E1 214.818} C_DIS
LIN {X -0.044,Y -142.321,Z 843.163,A 0.000,B 0.000,C 90.000,E1 209.283} C_DIS
LIN {X 0.077,Y -141.710,Z 843.152,A 0.000,B 0.000,C 90.000,E1 207.385} C_DIS
LIN {X -0.001,Y -139.471,Z 843.116,A 0.000,B 0.000,C 90.000,E1 200.918} C_DIS
LIN {X 0.053,Y -139.203,Z 843.106,A 0.000,B 0.000,C 90.000,E1 199.033} C_DIS
LIN {X -0.021,Y -138.329,Z 843.054,A 0.000,B 0.000,C 90.000,E1 189.726} C_DIS
LIN {X -0.018,Y -139.439,Z 843.007,A 0.000,B 0.000,C 90.000,E1 181.318} C_DIS
LIN {X 0.062,Y -140.973,Z 842.976,A 0.000,B 0.000,C 90.000,E1 175.698} C_DIS
LIN {X 0.012,Y -142.729,Z 842.956,A 0.000,B 0.000,C 90.000,E1 172.008} C_DIS
LIN {X -0.030,Y -145.114,Z 842.930,A 0.000,B 0.000,C 90.000,E1 167.409} C_DIS
LIN {X -0.036,Y -147.739,Z 842.910,A 0.000,B 0.000,C 90.000,E1 163.740} C_DIS
LIN {X 0.046,Y -150.403,Z 842.889,A 0.000,B 0.000,C 90.000,E1 160.061} C_DIS
LIN {X -0.080,Y -153.839,Z 842.869,A 0.000,B 0.000,C 90.000,E1 156.485} C_DIS
LIN {X -0.021,Y -157.249,Z 842.849,A 0.000,B 0.000,C 90.000,E1 152.871} C_DIS
LIN {X 0.057,Y -161.423,Z 842.829,A 0.000,B 0.000,C 90.000,E1 149.282} C_DIS
LIN {X -0.072,Y -165.624,Z 842.810,A 0.000,B 0.000,C 90.000,E1 145.801} C_DIS
LIN {X 0.048,Y -170.553,Z 842.790,A 0.000,B 0.000,C 90.000,E1 142.271} C_DIS
LIN {X -0.044,Y -175.432,Z 842.771,A 0.000,B 0.000,C 90.000,E1 138.852} C_DIS
LIN {X 0.073,Y -181.055,Z 842.752,A 0.000,B 0.000,C 90.000,E1 135.405} C_DIS
LIN {X -0.062,Y -186.491,Z 842.734,A 0.000,B 0.000,C 90.000,E1 132.081} C_DIS
LIN {X 0.007,Y -191.112,Z 842.720,A 0.000,B 0.000,C 90.000,E1 129.564} C_DIS
LIN {X 0.046,Y -192.918,Z 842.714,A 0.000,B 0.000,C 90.000,E1 128.463} C_DIS
LIN {X 0.021,Y -293.916,Z 842.714,A 0.000,B 0.000,C 90.000,E1 128.463} C_DIS
LIN {X -0.043,Y -298.225,Z 842.713,A 0.000,B 0.000,C 90.000,E1 128.338} C_DIS
LIN {X 0.077,Y -300.350,Z 842.712,A 0.000,B 0.000,C 90.000,E1 128.177} C_DIS
LIN {X 0.134,Y -303.258,Z 842.711,A 0.000,B 0.000,C 90.000,E1 127.890} C_DIS
LIN {X 0.053,Y -306.951,Z 842.708,A 0.000,B 0.000,C 90.000,E1 127.363} C_DIS
LIN {X 0.070,Y -308.512,Z 842.706,A 0.000,B 0.000,C 90.000,E1 127.030} C_DIS
LIN {X 0.027,Y -309.738,Z 842.704,A 0.000,B 0.000,C 90.000,E1 126.710} C_DIS
LIN {X -0.053,Y -320.834,Z 842.684,A 0.000,B 0.000,C 90.000,E1 123.166} C_DIS
LIN {X -0.202,Y -331.266,Z 842.668,A 0.000,B 0.000,C 90.000,E1 120.335} C_DIS
LIN {X -0.098,Y -343.047,Z 842.653,A 0.000,B 0.000,C 90.000,E1 117.513} C_DIS
LIN {X -0.134,Y -356.290,Z 842.638,A 0.000,B 0.000,C 90.000,E1 114.771} C_DIS
LIN {X 0.168,Y -369.377,Z 842.624,A 0.000,B 0.000,C 90.000,E1 112.333} C_DIS
LIN {X 0.183,Y -383.804,Z 842.611,A 0.000,B 0.000,C 90.000,E1 109.993} C_DIS
LIN {X -0.205,Y -399.670,Z 842.599,A 0.000,B 0.000,C 90.000,E1 107.764} C_DIS
LIN {X 0.181,Y -417.092,Z 842.586,A 0.000,B 0.000,C 90.000,E1 105.481} C_DIS
LIN {X -0.141,Y -436.190,Z 842.574,A 0.000,B 0.000,C 90.000,E1 103.355} C_DIS
LIN {X 0.051,Y -456.303,Z 842.563,A 0.000,B 0.000,C 90.000,E1 101.299} C_DIS
LIN {X -0.107,Y -466.567,Z 842.557,A 0.000,B 0.000,C 90.000,E1 100.366} C_DIS
LIN {X -0.148,Y -468.846,Z 842.556,A 0.000,B 0.000,C 90.000,E1 100.141} C_DIS
LIN {X -0.106,Y -470.567,Z 842.555,A 0.000,B 0.000,C 90.000,E1 99.905} C_DIS
LIN {X 0.211,Y -472.007,Z 842.554,A 0.000,B 0.000,C 90.000,E1 99.613} C_DIS
LIN {X 0.062,Y -473.081,Z 842.552,A 0.000,B 0.000,C 90.000,E1 99.378} C_DIS
LIN {X 0.171,Y -474.343,Z 842.549,A 0.000,B 0.000,C 90.000,E1 98.859} C_DIS
LIN {X -0.179,Y -474.595,Z 842.547,A 0.000,B 0.000,C 90.000,E1 98.398} C_DIS
LIN {X 0.014,Y -473.883,Z 842.544,A 0.000,B 0.000,C 90.000,E1 97.871} C_DIS
LIN {X 0.140,Y -472.093,Z 842.541,A 0.000,B 0.000,C 90.000,E1 97.352} C_DIS
LIN {X -0.062,Y -470.691,Z 842.540,A 0.000,B 0.000,C 90.000,E1 97.125} C_DIS
LIN {X -0.135,Y -454.512,Z 842.525,A 0.000,B 0.000,C 90.000,E1 94.588} C_DIS
LIN {X 0.025,Y -443.958,Z 842.515,A 0.000,B 0.000,C 90.000,E1 92.751} C_DIS
LIN {X -0.213,Y -434.630,Z 842.507,A 0.000,B 0.000,C 90.000,E1 91.203} C_DIS
LIN {X -0.184,Y -425.027,Z 842.498,A 0.000,B 0.000,C 90.000,E1 89.599} C_DIS
LIN {X 0.199,Y -413.582,Z 842.487,A 0.000,B 0.000,C 90.000,E1 87.650} C_DIS
LIN {X -0.135,Y -403.740,Z 842.478,A 0.000,B 0.000,C 90.000,E1 86.045} C_DIS
LIN {X -0.094,Y -390.666,Z 842.465,A 0.000,B 0.000,C 90.000,E1 83.799} C_DIS
LIN {X 0.046,Y -379.416,Z 842.454,A 0.000,B 0.000,C 90.000,E1 81.781} C_DIS
LIN {X 0.027,Y -365.296,Z 842.440,A 0.000,B 0.000,C 90.000,E1 79.162} C_DIS
LIN {X 0.136,Y -351.665,Z 842.425,A 0.000,B 0.000,C 90.000,E1 76.464} C_DIS
LIN {X 0.129,Y -341.082,Z 842.413,A 0.000,B 0.000,C 90.000,E1 74.338} C_DIS
LIN {X -0.076,Y -327.686,Z 842.398,A 0.000,B 0.000,C 90.000,E1 71.583} C_DIS
LIN {X 0.044,Y -316.072,Z 842.384,A 0.000,B 0.000,C 90.000,E1 69.028} C_DIS
LIN {X 0.018,Y -302.111,Z 842.366,A 0.000,B 0.000,C 90.000,E1 65.793} C_DIS
LIN {X -0.045,Y -290.006,Z 842.349,A 0.000,B 0.000,C 90.000,E1 62.820} C_DIS
LIN {X -0.120,Y -279.586,Z 842.334,A 0.000,B 0.000,C 90.000,E1 60.127} C_DIS
LIN {X 0.069,Y -267.019,Z 842.315,A 0.000,B 0.000,C 90.000,E1 56.628} C_DIS
LIN {X -0.018,Y -256.499,Z 842.297,A 0.000,B 0.000,C 90.000,E1 53.463} C_DIS
LIN {X 0.078,Y -245.553,Z 842.277,A 0.000,B 0.000,C 90.000,E1 49.828} C_DIS
LIN {X 0.110,Y -235.390,Z 842.256,A 0.000,B 0.000,C 90.000,E1 46.134} C_DIS
LIN {X -0.015,Y -226.039,Z 842.236,A 0.000,B 0.000,C 90.000,E1 42.405} C_DIS
LIN {X -0.068,Y -218.892,Z 842.219,A 0.000,B 0.000,C 90.000,E1 39.358} C_DIS
LIN {X 0.045,Y -210.503,Z 842.197,A 0.000,B 0.000,C 90.000,E1 35.438} C_DIS
LIN {X 0.090,Y -202.780,Z 842.175,A 0.000,B 0.000,C 90.000,E1 31.465} C_DIS
LIN {X -0.022,Y -197.233,Z 842.157,A 0.000,B 0.000,C 90.000,E1 28.281} C_DIS
LIN {X -0.022,Y -192.412,Z 842.139,A 0.000,B 0.000,C 90.000,E1 25.027} C_DIS
LIN {X 0.052,Y -188.369,Z 842.121,A 0.000,B 0.000,C 90.000,E1 21.716} C_DIS
LIN {X -0.008,Y -184.409,Z 842.098,A 0.000,B 0.000,C 90.000,E1 17.583} C_DIS
LIN {X 0.058,Y -181.222,Z 842.070,A 0.000,B 0.000,C 90.000,E1 12.535} C_DIS
LIN {X 0.068,Y -179.167,Z 842.028,A 0.000,B 0.000,C 90.000,E1 4.935} C_DIS
LIN {X -0.026,Y -180.857,Z 841.979,A 0.000,B 0.000,C 90.000,E1 356.159} C_DIS
LIN {X 0.053,Y -183.827,Z 841.951,A 0.000,B 0.000,C 90.000,E1 351.084} C_DIS
LIN {X -0.054,Y -187.293,Z 841.927,A 0.000,B 0.000,C 90.000,E1 346.937} C_DIS
LIN {X -0.016,Y -191.759,Z 841.904,A 0.000,B 0.000,C 90.000,E1 342.779} C_DIS
LIN {X 0.018,Y -197.079,Z 841.882,A 0.000,B 0.000,C 90.000,E1 338.666} C_DIS
LIN {X 0.108,Y -203.256,Z 841.859,A 0.000,B 0.000,C 90.000,E1 334.588} C_DIS
LIN {X 0.120,Y -210.247,Z 841.837,A 0.000,B 0.000,C 90.000,E1 330.589} C_DIS
LIN {X -0.078,Y -218.020,Z 841.815,A 0.000,B 0.000,C 90.000,E1 326.707} C_DIS
LIN {X 0.034,Y -224.864,Z 841.798,A 0.000,B 0.000,C 90.000,E1 323.577} C_DIS
LIN {X 0.000,Y -233.387,Z 841.779,A 0.000,B 0.000,C 90.000,E1 320.150} C_DIS
LIN {X -0.001,Y -242.762,Z 841.760,A 0.000,B 0.000,C 90.000,E1 316.782} C_DIS
LIN {X 0.088,Y -253.114,Z 841.742,A 0.000,B 0.000,C 90.000,E1 313.461} C_DIS
LIN {X -0.030,Y -264.424,Z 841.724,A 0.000,B 0.000,C 90.000,E1 310.253} C_DIS
LIN {X 0.043,Y -276.630,Z 841.706,A 0.000,B 0.000,C 90.000,E1 307.076} C_DIS
LIN {X 0.024,Y -289.990,Z 841.689,A 0.000,B 0.000,C 90.000,E1 303.992} C_DIS
LIN {X -0.088,Y -304.515,Z 841.672,A 0.000,B 0.000,C 90.000,E1 301.003} C_DIS
LIN {X 0.035,Y -316.880,Z 841.659,A 0.000,B 0.000,C 90.000,E1 298.693} C_DIS
LIN {X -0.045,Y -332.424,Z 841.645,A 0.000,B 0.000,C 90.000,E1 296.155} C_DIS
LIN {X -0.146,Y -353.698,Z 841.628,A 0.000,B 0.000,C 90.000,E1 293.078} C_DIS
LIN {X -0.104,Y -370.075,Z 841.616,A 0.000,B 0.000,C 90.000,E1 290.972} C_DIS
LIN {X -0.060,Y -395.290,Z 841.601,A 0.000,B 0.000,C 90.000,E1 288.127} C_DIS
LIN {X 0.160,Y -408.122,Z 841.593,A 0.000,B 0.000,C 90.000,E1 286.732} C_DIS
LIN {X -0.084,Y -420.774,Z 841.586,A 0.000,B 0.000,C 90.000,E1 285.426} C_DIS
LIN {X 0.091,Y -433.131,Z 841.578,A 0.000,B 0.000,C 90.000,E1 284.064} C_DIS
LIN {X 0.012,Y -442.756,Z 841.572,A 0.000,B 0.000,C 90.000,E1 283.008} C_DIS
LIN {X 0.048,Y -451.905,Z 841.566,A 0.000,B 0.000,C 90.000,E1 281.951} C_DIS
LIN {X 0.192,Y -460.411,Z 841.561,A 0.000,B 0.000,C 90.000,E1 280.894} C_DIS
LIN {X -0.108,Y -468.379,Z 841.555,A 0.000,B 0.000,C 90.000,E1 279.905} C_DIS
LIN {X -0.178,Y -473.875,Z 841.551,A 0.000,B 0.000,C 90.000,E1 279.151} C_DIS
LIN {X -0.204,Y -478.799,Z 841.547,A 0.000,B 0.000,C 90.000,E1 278.398} C_DIS
LIN {X -0.183,Y -482.981,Z 841.542,A 0.000,B 0.000,C 90.000,E1 277.644} C_DIS
LIN {X -0.131,Y -486.429,Z 841.538,A 0.000,B 0.000,C 90.000,E1 276.891} C_DIS
LIN {X 0.063,Y -488.376,Z 841.535,A 0.000,B 0.000,C 90.000,E1 276.372} C_DIS
LIN {X -0.222,Y -489.955,Z 841.533,A 0.000,B 0.000,C 90.000,E1 275.910} C_DIS
LIN {X -0.009,Y -491.201,Z 841.530,A 0.000,B 0.000,C 90.000,E1 275.391} C_DIS
LIN {X 0.169,Y -492.078,Z 841.527,A 0.000,B 0.000,C 90.000,E1 274.878} C_DIS
LIN {X -0.091,Y -492.565,Z 841.524,A 0.000,B 0.000,C 90.000,E1 274.416} C_DIS
LIN {X 0.141,Y -492.726,Z 841.522,A 0.000,B 0.000,C 90.000,E1 273.898} C_DIS
LIN {X -0.148,Y -492.505,Z 841.519,A 0.000,B 0.000,C 90.000,E1 273.440} C_DIS
LIN {X 0.084,Y -491.891,Z 841.516,A 0.000,B 0.000,C 90.000,E1 272.922} C_DIS
LIN {X -0.201,Y -490.842,Z 841.514,A 0.000,B 0.000,C 90.000,E1 272.465} C_DIS
LIN {X 0.004,Y -489.358,Z 841.511,A 0.000,B 0.000,C 90.000,E1 271.949} C_DIS
LIN {X 0.217,Y -487.407,Z 841.508,A 0.000,B 0.000,C 90.000,E1 271.432} C_DIS
LIN {X -0.081,Y -484.866,Z 841.505,A 0.000,B 0.000,C 90.000,E1 270.974} C_DIS
LIN {X 0.090,Y -481.719,Z 841.503,A 0.000,B 0.000,C 90.000,E1 270.458} C_DIS
LIN {X -0.234,Y -477.902,Z 841.500,A 0.000,B 0.000,C 90.000,E1 270.000} C_DIS
LIN {X -0.098,Y -473.205,Z 841.497,A 0.000,B 0.000,C 90.000,E1 269.484} C_DIS
LIN {X 0.221,Y -470.603,Z 841.496,A 0.000,B 0.000,C 90.000,E1 269.198} C_DIS
LIN {X 0.148,Y -464.794,Z 841.493,A 0.000,B 0.000,C 90.000,E1 268.740} C_DIS
LIN {X 0.088,Y -458.393,Z 841.491,A 0.000,B 0.000,C 90.000,E1 268.339} C_DIS
LIN {X 0.085,Y -451.489,Z 841.489,A 0.000,B 0.000,C 90.000,E1 267.993} C_DIS
LIN {X 0.147,Y -443.990,Z 841.487,A 0.000,B 0.000,C 90.000,E1 267.707} C_DIS
LIN {X -0.173,Y -436.026,Z 841.486,A 0.000,B 0.000,C 90.000,E1 267.535} C_DIS
LIN {X -0.049,Y -427.018,Z 841.485,A 0.000,B 0.000,C 90.000,E1 267.364} C_DIS
LIN {X -0.096,Y -421.017,Z 841.485,A 0.000,B 0.000,C 90.000,E1 267.306} C_DIS
LIN {X 0.175,Y -416.588,Z 841.485,A 0.000,B 0.000,C 90.000,E1 267.249} C_DIS
LIN {X 0.045,Y -181.020,Z 841.485,A 0.000,B 0.000,C 90.000,E1 267.249} C_DIS
LIN {X 0.062,Y -180.761,Z 841.470,A 0.000,B 0.000,C 90.000,E1 264.666} C_DIS
LIN {X -0.046,Y -178.856,Z 841.442,A 0.000,B 0.000,C 90.000,E1 259.634} C_DIS
LIN {X 0.025,Y -175.898,Z 841.414,A 0.000,B 0.000,C 90.000,E1 254.519} C_DIS
LIN {X -0.035,Y -174.575,Z 841.405,A 0.000,B 0.000,C 90.000,E1 252.834} C_DIS
LIN {X 0.000,Y -171.559,Z 841.381,A 0.000,B 0.000,C 90.000,E1 248.539} C_DIS
LIN {X 0.055,Y -167.783,Z 841.357,A 0.000,B 0.000,C 90.000,E1 244.204} C_DIS
LIN {X -0.003,Y -166.496,Z 841.347,A 0.000,B 0.000,C 90.000,E1 242.487} C_DIS
LIN {X -0.007,Y -163.206,Z 841.328,A 0.000,B 0.000,C 90.000,E1 238.997} C_DIS
LIN {X -0.043,Y -161.170,Z 841.313,A 0.000,B 0.000,C 90.000,E1 236.373} C_DIS
LIN {X 0.081,Y -157.185,Z 841.289,A 0.000,B 0.000,C 90.000,E1 231.904} C_DIS
LIN {X 0.004,Y -155.915,Z 841.279,A 0.000,B 0.000,C 90.000,E1 230.150} C_DIS
LIN {X 0.061,Y -152.165,Z 841.254,A 0.000,B 0.000,C 90.000,E1 225.648} C_DIS
LIN {X -0.030,Y -150.414,Z 841.239,A 0.000,B 0.000,C 90.000,E1 222.975} C_DIS
LIN {X 0.012,Y -147.143,Z 841.213,A 0.000,B 0.000,C 90.000,E1 218.418} C_DIS
LIN {X 0.008,Y -145.701,Z 841.198,A 0.000,B 0.000,C 90.000,E1 215.678} C_DIS
LIN {X 0.016,Y -143.085,Z 841.173,A 0.000,B 0.000,C 90.000,E1 211.082} C_DIS
LIN {X 0.021,Y -141.702,Z 841.152,A 0.000,B 0.000,C 90.000,E1 207.385} C_DIS
LIN {X -0.056,Y -139.467,Z 841.116,A 0.000,B 0.000,C 90.000,E1 200.918} C_DIS
LIN {X -0.002,Y -139.200,Z 841.106,A 0.000,B 0.000,C 90.000,E1 199.033} C_DIS
LIN {X 0.061,Y -138.327,Z 841.054,A 0.000,B 0.000,C 90.000,E1 189.670} C_DIS
LIN {X 0.066,Y -139.444,Z 841.007,A 0.000,B 0.000,C 90.000,E1 181.260} C_DIS
LIN {X 0.007,Y -140.982,Z 840.976,A 0.000,B 0.000,C 90.000,E1 175.698} C_DIS
LIN {X -0.043,Y -142.737,Z 840.956,A 0.000,B 0.000,C 90.000,E1 172.008} C_DIS
LIN {X 0.055,Y -145.129,Z 840.930,A 0.000,B 0.000,C 90.000,E1 167.353} C_DIS
LIN {X 0.049,Y -147.752,Z 840.909,A 0.000,B 0.000,C 90.000,E1 163.685} C_DIS
LIN {X -0.012,Y -150.421,Z 840.889,A 0.000,B 0.000,C 90.000,E1 160.061} C_DIS
LIN {X 0.003,Y -153.862,Z 840.869,A 0.000,B 0.000,C 90.000,E1 156.433} C_DIS
LIN {X -0.080,Y -157.273,Z 840.849,A 0.000,B 0.000,C 90.000,E1 152.871} C_DIS
LIN {X -0.003,Y -161.451,Z 840.829,A 0.000,B 0.000,C 90.000,E1 149.282} C_DIS
LIN {X 0.003,Y -165.651,Z 840.810,A 0.000,B 0.000,C 90.000,E1 145.754} C_DIS
LIN {X -0.014,Y -170.586,Z 840.790,A 0.000,B 0.000,C 90.000,E1 142.271} C_DIS
LIN {X -0.107,Y -175.463,Z 840.771,A 0.000,B 0.000,C 90.000,E1 138.852} C_DIS
LIN {X 0.008,Y -181.086,Z 840.752,A 0.000,B 0.000,C 90.000,E1 135.405} C_DIS
LIN {X -0.002,Y -186.527,Z 840.734,A 0.000,B 0.000,C 90.000,E1 132.043} C_DIS
LIN {X -0.060,Y -191.144,Z 840.720,A 0.000,B 0.000,C 90.000,E1 129.564} C_DIS
LIN {X 0.076,Y -192.903,Z 840.714,A 0.000,B 0.000,C 90.000,E1 128.463} C_DIS
LIN {X 0.067,Y -293.628,Z 840.714,A 0.000,B 0.000,C 90.000,E1 128.463} C_DIS
LIN {X -0.081,Y -295.331,Z 840.714,A 0.000,B 0.000,C 90.000,E1 128.463} C_DIS
LIN {X -0.027,Y -300.647,Z 840.712,A 0.000,B 0.000,C 90.000,E1 128.177} C_DIS
LIN {X 0.029,Y -303.448,Z 840.711,A 0.000,B 0.000,C 90.000,E1 127.890} C_DIS
LIN {X 0.102,Y -307.139,Z 840.707,A 0.000,B 0.000,C 90.000,E1 127.317} C_DIS
LIN {X 0.061,Y -308.651,Z 840.706,A 0.000,B 0.000,C 90.000,E1 126.996} C_DIS
LIN {X 0.080,Y -309.838,Z 840.704,A 0.000,B 0.000,C 90.000,E1 126.664} C_DIS
LIN {X 0.191,Y -320.934,Z 840.684,A 0.000,B 0.000,C 90.000,E1 123.086} C_DIS
LIN {X 0.048,Y -331.381,Z 840.668,A 0.000,B 0.000,C 90.000,E1 120.256} C_DIS
LIN {X 0.000,Y -343.180,Z 840.653,A 0.000,B 0.000,C 90.000,E1 117.462} C_DIS
LIN {X -0.020,Y -356.441,Z 840.637,A 0.000,B 0.000,C 90.000,E1 114.719} C_DIS
LIN {X -0.046,Y -369.547,Z 840.624,A 0.000,B 0.000,C 90.000,E1 112.333} C_DIS
LIN {X -0.035,Y -383.991,Z 840.611,A 0.000,B 0.000,C 90.000,E1 109.993} C_DIS
LIN {X 0.075,Y -399.879,Z 840.598,A 0.000,B 0.000,C 90.000,E1 107.692} C_DIS
LIN {X -0.046,Y -417.324,Z 840.586,A 0.000,B 0.000,C 90.000,E1 105.481} C_DIS
LIN {X 0.055,Y -436.442,Z 840.574,A 0.000,B 0.000,C 90.000,E1 103.300} C_DIS
LIN {X -0.169,Y -456.563,Z 840.563,A 0.000,B 0.000,C 90.000,E1 101.299} C_DIS
LIN {X 0.136,Y -466.832,Z 840.557,A 0.000,B 0.000,C 90.000,E1 100.310} C_DIS
LIN {X 0.181,Y -469.051,Z 840.556,A 0.000,B 0.000,C 90.000,E1 100.074} C_DIS
LIN {X 0.145,Y -470.729,Z 840.555,A 0.000,B 0.000,C 90.000,E1 99.849} C_DIS
LIN {X -0.003,Y -472.137,Z 840.553,A 0.000,B 0.000,C 90.000,E1 99.613} C_DIS
LIN {X -0.152,Y -473.184,Z 840.552,A 0.000,B 0.000,C 90.000,E1 99.378} C_DIS
LIN {X -0.042,Y -474.401,Z 840.549,A 0.000,B 0.000,C 90.000,E1 98.859} C_DIS
LIN {X 0.077,Y -474.614,Z 840.546,A 0.000,B 0.000,C 90.000,E1 98.341} C_DIS
LIN {X -0.198,Y -473.862,Z 840.544,A 0.000,B 0.000,C 90.000,E1 97.871} C_DIS
LIN {X -0.071,Y -472.023,Z 840.541,A 0.000,B 0.000,C 90.000,E1 97.352} C_DIS
LIN {X 0.053,Y -468.911,Z 840.538,A 0.000,B 0.000,C 90.000,E1 96.834} C_DIS
LIN {X 0.112,Y -454.402,Z 840.525,A 0.000,B 0.000,C 90.000,E1 94.531} C_DIS
LIN {X -0.177,Y -443.822,Z 840.515,A 0.000,B 0.000,C 90.000,E1 92.751} C_DIS
LIN {X 0.019,Y -434.521,Z 840.506,A 0.000,B 0.000,C 90.000,E1 91.146} C_DIS
LIN {X 0.042,Y -424.922,Z 840.497,A 0.000,B 0.000,C 90.000,E1 89.542} C_DIS
LIN {X 0.003,Y -413.464,Z 840.487,A 0.000,B 0.000,C 90.000,E1 87.650} C_DIS
LIN {X 0.075,Y -403.612,Z 840.478,A 0.000,B 0.000,C 90.000,E1 85.988} C_DIS
LIN {X 0.104,Y -390.520,Z 840.465,A 0.000,B 0.000,C 90.000,E1 83.742} C_DIS
LIN {X -0.141,Y -379.274,Z 840.454,A 0.000,B 0.000,C 90.000,E1 81.781} C_DIS
LIN {X -0.156,Y -365.150,Z 840.440,A 0.000,B 0.000,C 90.000,E1 79.162} C_DIS
LIN {X -0.044,Y -351.558,Z 840.425,A 0.000,B 0.000,C 90.000,E1 76.464} C_DIS
LIN {X -0.049,Y -341.016,Z 840.413,A 0.000,B 0.000,C 90.000,E1 74.338} C_DIS
LIN {X -0.117,Y -329.114,Z 840.399,A 0.000,B 0.000,C 90.000,E1 71.873} C_DIS
LIN {X -0.063,Y -317.477,Z 840.385,A 0.000,B 0.000,C 90.000,E1 69.337} C_DIS
LIN {X -0.042,Y -303.481,Z 840.367,A 0.000,B 0.000,C 90.000,E1 66.102} C_DIS
LIN {X -0.052,Y -292.698,Z 840.352,A 0.000,B 0.000,C 90.000,E1 63.461} C_DIS
LIN {X 0.048,Y -282.264,Z 840.338,A 0.000,B 0.000,C 90.000,E1 60.745} C_DIS
LIN {X -0.001,Y -270.863,Z 840.320,A 0.000,B 0.000,C 90.000,E1 57.661} C_DIS
LIN {X 0.127,Y -259.024,Z 840.301,A 0.000,B 0.000,C 90.000,E1 54.116} C_DIS
LIN {X -0.054,Y -247.957,Z 840.281,A 0.000,B 0.000,C 90.000,E1 50.561} C_DIS
LIN {X 0.076,Y -237.645,Z 840.260,A 0.000,B 0.000,C 90.000,E1 46.863} C_DIS
LIN {X 0.007,Y -228.164,Z 840.240,A 0.000,B 0.000,C 90.000,E1 43.137} C_DIS
LIN {X -0.001,Y -220.926,Z 840.223,A 0.000,B 0.000,C 90.000,E1 40.092} C_DIS
LIN {X 0.003,Y -212.406,Z 840.201,A 0.000,B 0.000,C 90.000,E1 36.217} C_DIS
LIN {X -0.065,Y -206.090,Z 840.184,A 0.000,B 0.000,C 90.000,E1 33.086} C_DIS
LIN {X 0.010,Y -200.216,Z 840.166,A 0.000,B 0.000,C 90.000,E1 29.873} C_DIS
LIN {X 0.089,Y -195.011,Z 840.148,A 0.000,B 0.000,C 90.000,E1 26.616} C_DIS
LIN {X -0.047,Y -190.589,Z 840.130,A 0.000,B 0.000,C 90.000,E1 23.387} C_DIS
LIN {X -0.090,Y -186.156,Z 840.107,A 0.000,B 0.000,C 90.000,E1 19.268} C_DIS
LIN {X 0.017,Y -182.916,Z 840.084,A 0.000,B 0.000,C 90.000,E1 15.064} C_DIS
LIN {X -0.074,Y -180.276,Z 840.051,A 0.000,B 0.000,C 90.000,E1 9.208} C_DIS
LIN {X -0.018,Y -181.164,Z 839.979,A 0.000,B 0.000,C 90.000,E1 356.159} C_DIS
LIN {X 0.073,Y -184.147,Z 839.951,A 0.000,B 0.000,C 90.000,E1 351.084} C_DIS
LIN {X -0.024,Y -187.627,Z 839.927,A 0.000,B 0.000,C 90.000,E1 346.937} C_DIS
LIN {X 0.025,Y -192.055,Z 839.904,A 0.000,B 0.000,C 90.000,E1 342.779} C_DIS
LIN {X -0.114,Y -197.349,Z 839.882,A 0.000,B 0.000,C 90.000,E1 338.720} C_DIS
LIN {X -0.102,Y -203.478,Z 839.859,A 0.000,B 0.000,C 90.000,E1 334.665} C_DIS
LIN {X 0.000,Y -209.020,Z 839.841,A 0.000,B 0.000,C 90.000,E1 331.435} C_DIS
LIN {X -0.049,Y -216.626,Z 839.819,A 0.000,B 0.000,C 90.000,E1 327.502} C_DIS
LIN {X -0.091,Y -223.310,Z 839.802,A 0.000,B 0.000,C 90.000,E1 324.402} C_DIS
LIN {X -0.076,Y -230.634,Z 839.785,A 0.000,B 0.000,C 90.000,E1 321.331} C_DIS
LIN {X 0.016,Y -239.740,Z 839.766,A 0.000,B 0.000,C 90.000,E1 317.919} C_DIS
LIN {X 0.020,Y -249.744,Z 839.748,A 0.000,B 0.000,C 90.000,E1 314.595} C_DIS
LIN {X -0.039,Y -260.694,Z 839.730,A 0.000,B 0.000,C 90.000,E1 311.353} C_DIS
LIN {X -0.086,Y -272.556,Z 839.712,A 0.000,B 0.000,C 90.000,E1 308.177} C_DIS
LIN {X 0.108,Y -285.417,Z 839.695,A 0.000,B 0.000,C 90.000,E1 305.025} C_DIS
LIN {X 0.031,Y -301.116,Z 839.676,A 0.000,B 0.000,C 90.000,E1 301.671} C_DIS
LIN {X -0.139,Y -314.958,Z 839.661,A 0.000,B 0.000,C 90.000,E1 299.077} C_DIS
LIN {X 0.065,Y -328.268,Z 839.649,A 0.000,B 0.000,C 90.000,E1 296.796} C_DIS
LIN {X -0.022,Y -349.063,Z 839.632,A 0.000,B 0.000,C 90.000,E1 293.695} C_DIS
LIN {X -0.081,Y -364.960,Z 839.620,A 0.000,B 0.000,C 90.000,E1 291.589} C_DIS
LIN {X 0.037,Y -382.205,Z 839.608,A 0.000,B 0.000,C 90.000,E1 289.523} C_DIS
LIN {X 0.078,Y -399.997,Z 839.598,A 0.000,B 0.000,C 90.000,E1 287.583} C_DIS
LIN {X -0.161,Y -412.815,Z 839.590,A 0.000,B 0.000,C 90.000,E1 286.260} C_DIS
LIN {X -0.056,Y -425.429,Z 839.583,A 0.000,B 0.000,C 90.000,E1 284.898} C_DIS
LIN {X 0.123,Y -437.683,Z 839.575,A 0.000,B 0.000,C 90.000,E1 283.536} C_DIS
LIN {X 0.100,Y -447.138,Z 839.569,A 0.000,B 0.000,C 90.000,E1 282.479} C_DIS
LIN {X 0.189,Y -455.979,Z 839.564,A 0.000,B 0.000,C 90.000,E1 281.422} C_DIS
LIN {X -0.075,Y -464.244,Z 839.558,A 0.000,B 0.000,C 90.000,E1 280.423} C_DIS
LIN {X 0.123,Y -471.892,Z 839.552,A 0.000,B 0.000,C 90.000,E1 279.378} C_DIS
LIN {X 0.085,Y -477.004,Z 839.548,A 0.000,B 0.000,C 90.000,E1 278.624} C_DIS
LIN {X 0.217,Y -480.084,Z 839.545,A 0.000,B 0.000,C 90.000,E1 278.106} C_DIS
LIN {X 0.247,Y -484.071,Z 839.541,A 0.000,B 0.000,C 90.000,E1 277.352} C_DIS
LIN {X -0.056,Y -486.295,Z 839.538,A 0.000,B 0.000,C 90.000,E1 276.891} C_DIS
LIN {X 0.138,Y -488.247,Z 839.535,A 0.000,B 0.000,C 90.000,E1 276.372} C_DIS
LIN {X -0.147,Y -489.871,Z 839.533,A 0.000,B 0.000,C 90.000,E1 275.910} C_DIS
LIN {X 0.064,Y -491.098,Z 839.530,A 0.000,B 0.000,C 90.000,E1 275.391} C_DIS
LIN {X -0.248,Y -492.020,Z 839.527,A 0.000,B 0.000,C 90.000,E1 274.935} C_DIS
LIN {X -0.019,Y -492.549,Z 839.525,A 0.000,B 0.000,C 90.000,E1 274.416} C_DIS
LIN {X 0.213,Y -492.720,Z 839.522,A 0.000,B 0.000,C 90.000,E1 273.898} C_DIS
LIN {X -0.075,Y -492.507,Z 839.519,A 0.000,B 0.000,C 90.000,E1 273.440} C_DIS
LIN {X 0.156,Y -491.927,Z 839.516,A 0.000,B 0.000,C 90.000,E1 272.922} C_DIS
LIN {X -0.129,Y -490.916,Z 839.514,A 0.000,B 0.000,C 90.000,E1 272.465} C_DIS
LIN {X 0.076,Y -489.465,Z 839.511,A 0.000,B 0.000,C 90.000,E1 271.949} C_DIS
LIN {X -0.198,Y -487.550,Z 839.508,A 0.000,B 0.000,C 90.000,E1 271.489} C_DIS
LIN {X -0.008,Y -485.070,Z 839.505,A 0.000,B 0.000,C 90.000,E1 270.974} C_DIS
LIN {X 0.164,Y -481.934,Z 839.503,A 0.000,B 0.000,C 90.000,E1 270.458} C_DIS
LIN {X -0.160,Y -478.188,Z 839.500,A 0.000,B 0.000,C 90.000,E1 270.000} C_DIS
LIN {X -0.024,Y -473.574,Z 839.497,A 0.000,B 0.000,C 90.000,E1 269.484} C_DIS
LIN {X -0.204,Y -470.939,Z 839.496,A 0.000,B 0.000,C 90.000,E1 269.255} C_DIS
LIN {X 0.134,Y -465.110,Z 839.493,A 0.000,B 0.000,C 90.000,E1 268.740} C_DIS
LIN {X 0.015,Y -458.717,Z 839.491,A 0.000,B 0.000,C 90.000,E1 268.339} C_DIS
LIN {X -0.030,Y -451.782,Z 839.489,A 0.000,B 0.000,C 90.000,E1 267.993} C_DIS
LIN {X 0.006,Y -444.196,Z 839.487,A 0.000,B 0.000,C 90.000,E1 267.707} C_DIS
LIN {X 0.103,Y -436.319,Z 839.486,A 0.000,B 0.000,C 90.000,E1 267.478} C_DIS
LIN {X -0.208,Y -427.460,Z 839.485,A 0.000,B 0.000,C 90.000,E1 267.364} C_DIS
LIN {X 0.032,Y -417.812,Z 839.485,A 0.000,B 0.000,C 90.000,E1 267.249} C_DIS
LIN {X -0.017,Y -181.018,Z 839.485,A 0.000,B 0.000,C 90.000,E1 267.249} C_DIS
LIN {X -0.058,Y -180.908,Z 839.475,A 0.000,B 0.000,C 90.000,E1 265.527} C_DIS
LIN {X -0.001,Y -180.753,Z 839.470,A 0.000,B 0.000,C 90.000,E1 264.666} C_DIS
LIN {X 0.068,Y -178.846,Z 839.442,A 0.000,B 0.000,C 90.000,E1 259.577} C_DIS
LIN {X -0.037,Y -175.889,Z 839.414,A 0.000,B 0.000,C 90.000,E1 254.519} C_DIS
LIN {X 0.070,Y -174.559,Z 839.404,A 0.000,B 0.000,C 90.000,E1 252.779} C_DIS
LIN {X -0.061,Y -171.543,Z 839.381,A 0.000,B 0.000,C 90.000,E1 248.539} C_DIS
LIN {X -0.004,Y -167.767,Z 839.357,A 0.000,B 0.000,C 90.000,E1 244.204} C_DIS
LIN {X -0.064,Y -166.476,Z 839.347,A 0.000,B 0.000,C 90.000,E1 242.487} C_DIS
LIN {X -0.067,Y -163.189,Z 839.328,A 0.000,B 0.000,C 90.000,E1 238.997} C_DIS
LIN {X -0.012,Y -161.150,Z 839.313,A 0.000,B 0.000,C 90.000,E1 236.342} C_DIS
LIN {X 0.024,Y -157.168,Z 839.288,A 0.000,B 0.000,C 90.000,E1 231.904} C_DIS
LIN {X -0.053,Y -155.900,Z 839.279,A 0.000,B 0.000,C 90.000,E1 230.150} C_DIS
LIN {X 0.005,Y -152.150,Z 839.254,A 0.000,B 0.000,C 90.000,E1 225.648} C_DIS
LIN {X 0.024,Y -150.400,Z 839.239,A 0.000,B 0.000,C 90.000,E1 222.933} C_DIS
LIN {X 0.047,Y -147.130,Z 839.213,A 0.000,B 0.000,C 90.000,E1 218.382} C_DIS
LIN {X -0.046,Y -145.692,Z 839.198,A 0.000,B 0.000,C 90.000,E1 215.678} C_DIS
LIN {X 0.036,Y -143.074,Z 839.173,A 0.000,B 0.000,C 90.000,E1 211.052} C_DIS
LIN {X -0.033,Y -141.694,Z 839.152,A 0.000,B 0.000,C 90.000,E1 207.385} C_DIS
LIN {X 0.021,Y -139.463,Z 839.116,A 0.000,B 0.000,C 90.000,E1 200.865} C_DIS
LIN {X -0.056,Y -139.197,Z 839.106,A 0.000,B 0.000,C 90.000,E1 199.033} C_DIS
LIN {X 0.007,Y -138.325,Z 839.054,A 0.000,B 0.000,C 90.000,E1 189.670} C_DIS
LIN {X 0.013,Y -139.449,Z 839.007,A 0.000,B 0.000,C 90.000,E1 181.260} C_DIS
LIN {X -0.047,Y -140.991,Z 838.976,A 0.000,B 0.000,C 90.000,E1 175.698} C_DIS
LIN {X 0.044,Y -142.746,Z 838.955,A 0.000,B 0.000,C 90.000,E1 171.951} C_DIS
LIN {X 0.000,Y -145.143,Z 838.930,A 0.000,B 0.000,C 90.000,E1 167.353} C_DIS
LIN {X -0.007,Y -147.765,Z 838.909,A 0.000,B 0.000,C 90.000,E1 163.685} C_DIS
LIN {X -0.068,Y -150.439,Z 838.889,A 0.000,B 0.000,C 90.000,E1 160.061} C_DIS
LIN {X 0.008,Y -153.885,Z 838.869,A 0.000,B 0.000,C 90.000,E1 156.410} C_DIS
LIN {X 0.002,Y -157.295,Z 838.849,A 0.000,B 0.000,C 90.000,E1 152.820} C_DIS
LIN {X 0.021,Y -161.479,Z 838.829,A 0.000,B 0.000,C 90.000,E1 149.253} C_DIS
LIN {X 0.038,Y -165.678,Z 838.810,A 0.000,B 0.000,C 90.000,E1 145.722} C_DIS
LIN {X -0.076,Y -170.618,Z 838.790,A 0.000,B 0.000,C 90.000,E1 142.271} C_DIS
LIN {X 0.078,Y -175.494,Z 838.771,A 0.000,B 0.000,C 90.000,E1 138.771} C_DIS
LIN {X -0.055,Y -181.115,Z 838.752,A 0.000,B 0.000,C 90.000,E1 135.405} C_DIS
LIN {X 0.072,Y -186.562,Z 838.733,A 0.000,B 0.000,C 90.000,E1 132.000} C_DIS
LIN {X 0.022,Y -191.176,Z 838.720,A 0.000,B 0.000,C 90.000,E1 129.519} C_DIS
LIN {X 0.081,Y -192.901,Z 838.714,A 0.000,B 0.000,C 90.000,E1 128.463} C_DIS
LIN {X 0.088,Y -293.859,Z 838.714,A 0.000,B 0.000,C 90.000,E1 128.463} C_DIS
LIN {X -0.180,Y -296.179,Z 838.714,A 0.000,B 0.000,C 90.000,E1 128.463} C_DIS
LIN {X -0.129,Y -300.924,Z 838.712,A 0.000,B 0.000,C 90.000,E1 128.177} C_DIS
LIN {X -0.074,Y -303.628,Z 838.710,A 0.000,B 0.000,C 90.000,E1 127.890} C_DIS
LIN {X -0.086,Y -307.313,Z 838.707,A 0.000,B 0.000,C 90.000,E1 127.317} C_DIS
LIN {X 0.119,Y -308.778,Z 838.705,A 0.000,B 0.000,C 90.000,E1 126.950} C_DIS
LIN {X -0.109,Y -309.929,Z 838.704,A 0.000,B 0.000,C 90.000,E1 126.664} C_DIS
LIN {X -0.071,Y -319.944,Z 838.686,A 0.000,B 0.000,C 90.000,E1 123.420} C_DIS
LIN {X 0.035,Y -330.259,Z 838.670,A 0.000,B 0.000,C 90.000,E1 120.541} C_DIS
LIN {X 0.118,Y -341.922,Z 838.654,A 0.000,B 0.000,C 90.000,E1 117.719} C_DIS
LIN {X 0.071,Y -355.028,Z 838.639,A 0.000,B 0.000,C 90.000,E1 114.975} C_DIS
LIN {X 0.016,Y -367.990,Z 838.625,A 0.000,B 0.000,C 90.000,E1 112.589} C_DIS
LIN {X -0.003,Y -382.279,Z 838.612,A 0.000,B 0.000,C 90.000,E1 110.248} C_DIS
LIN {X 0.074,Y -397.999,Z 838.600,A 0.000,B 0.000,C 90.000,E1 107.946} C_DIS
LIN {X 0.031,Y -415.263,Z 838.587,A 0.000,B 0.000,C 90.000,E1 105.717} C_DIS
LIN {X 0.079,Y -434.189,Z 838.575,A 0.000,B 0.000,C 90.000,E1 103.536} C_DIS
LIN {X 0.146,Y -454.244,Z 838.564,A 0.000,B 0.000,C 90.000,E1 101.478} C_DIS
LIN {X -0.066,Y -467.076,Z 838.557,A 0.000,B 0.000,C 90.000,E1 100.310} C_DIS
LIN {X -0.048,Y -469.266,Z 838.556,A 0.000,B 0.000,C 90.000,E1 100.074} C_DIS
LIN {X -0.112,Y -470.921,Z 838.555,A 0.000,B 0.000,C 90.000,E1 99.849} C_DIS
LIN {X 0.207,Y -472.288,Z 838.553,A 0.000,B 0.000,C 90.000,E1 99.557} C_DIS
LIN {X 0.059,Y -473.301,Z 838.552,A 0.000,B 0.000,C 90.000,E1 99.321} C_DIS
LIN {X 0.171,Y -474.464,Z 838.549,A 0.000,B 0.000,C 90.000,E1 98.803} C_DIS
LIN {X -0.177,Y -474.629,Z 838.546,A 0.000,B 0.000,C 90.000,E1 98.341} C_DIS
LIN {X 0.017,Y -473.825,Z 838.543,A 0.000,B 0.000,C 90.000,E1 97.814} C_DIS
LIN {X 0.144,Y -471.923,Z 838.541,A 0.000,B 0.000,C 90.000,E1 97.296} C_DIS
LIN {X -0.199,Y -468.771,Z 838.538,A 0.000,B 0.000,C 90.000,E1 96.834} C_DIS
LIN {X 0.098,Y -455.801,Z 838.526,A 0.000,B 0.000,C 90.000,E1 94.759} C_DIS
LIN {X 0.021,Y -443.671,Z 838.515,A 0.000,B 0.000,C 90.000,E1 92.694} C_DIS
LIN {X 0.212,Y -434.377,Z 838.506,A 0.000,B 0.000,C 90.000,E1 91.088} C_DIS
LIN {X -0.197,Y -424.777,Z 838.497,A 0.000,B 0.000,C 90.000,E1 89.542} C_DIS
LIN {X 0.180,Y -413.311,Z 838.487,A 0.000,B 0.000,C 90.000,E1 87.593} C_DIS
LIN {X -0.158,Y -403.451,Z 838.478,A 0.000,B 0.000,C 90.000,E1 85.988} C_DIS
LIN {X -0.125,Y -390.352,Z 838.465,A 0.000,B 0.000,C 90.000,E1 83.742} C_DIS
LIN {X 0.008,Y -379.108,Z 838.454,A 0.000,B 0.000,C 90.000,E1 81.724} C_DIS
LIN {X -0.020,Y -364.986,Z 838.439,A 0.000,B 0.000,C 90.000,E1 79.106} C_DIS
LIN {X 0.133,Y -352.906,Z 838.426,A 0.000,B 0.000,C 90.000,E1 76.700} C_DIS
LIN {X 0.157,Y -342.425,Z 838.414,A 0.000,B 0.000,C 90.000,E1 74.574} C_DIS
LIN {X 0.015,Y -330.514,Z 838.401,A 0.000,B 0.000,C 90.000,E1 72.127} C_DIS
LIN {X -0.095,Y -318.882,Z 838.387,A 0.000,B 0.000,C 90.000,E1 69.625} C_DIS
LIN {X 0.041,Y -303.465,Z 838.367,A 0.000,B 0.000,C 90.000,E1 66.049} C_DIS
LIN {X 0.018,Y -291.394,Z 838.350,A 0.000,B 0.000,C 90.000,E1 63.076} C_DIS
LIN {X -0.024,Y -281.054,Z 838.335,A 0.000,B 0.000,C 90.000,E1 60.383} C_DIS
LIN {X 0.134,Y -269.797,Z 838.318,A 0.000,B 0.000,C 90.000,E1 57.248} C_DIS
LIN {X 0.016,Y -258.112,Z 838.299,A 0.000,B 0.000,C 90.000,E1 53.749} C_DIS
LIN {X -0.007,Y -248.209,Z 838.281,A 0.000,B 0.000,C 90.000,E1 50.517} C_DIS
LIN {X -0.054,Y -237.901,Z 838.260,A 0.000,B 0.000,C 90.000,E1 46.863} C_DIS
LIN {X 0.056,Y -228.428,Z 838.240,A 0.000,B 0.000,C 90.000,E1 43.095} C_DIS
LIN {X -0.108,Y -221.197,Z 838.223,A 0.000,B 0.000,C 90.000,E1 40.092} C_DIS
LIN {X 0.079,Y -212.674,Z 838.201,A 0.000,B 0.000,C 90.000,E1 36.171} C_DIS
LIN {X 0.022,Y -206.368,Z 838.184,A 0.000,B 0.000,C 90.000,E1 33.038} C_DIS
LIN {X -0.066,Y -200.496,Z 838.166,A 0.000,B 0.000,C 90.000,E1 29.873} C_DIS
LIN {X 0.021,Y -195.287,Z 838.148,A 0.000,B 0.000,C 90.000,E1 26.616} C_DIS
LIN {X 0.069,Y -190.865,Z 838.130,A 0.000,B 0.000,C 90.000,E1 23.334} C_DIS
LIN {X 0.036,Y -186.469,Z 838.107,A 0.000,B 0.000,C 90.000,E1 19.214} C_DIS
LIN {X -0.022,Y -183.208,Z 838.084,A 0.000,B 0.000,C 90.000,E1 15.064} C_DIS
LIN {X 0.078,Y -180.556,Z 838.051,A 0.000,B 0.000,C 90.000,E1 9.151} C_DIS
LIN {X -0.010,Y -181.476,Z 837.979,A 0.000,B 0.000,C 90.000,E1 356.159} C_DIS
LIN {X -0.090,Y -184.457,Z 837.951,A 0.000,B 0.000,C 90.000,E1 351.141} C_DIS
LIN {X 0.005,Y -187.937,Z 837.927,A 0.000,B 0.000,C 90.000,E1 346.937} C_DIS
LIN {X 0.064,Y -192.352,Z 837.904,A 0.000,B 0.000,C 90.000,E1 342.779} C_DIS
LIN {X -0.064,Y -197.612,Z 837.882,A 0.000,B 0.000,C 90.000,E1 338.720} C_DIS
LIN {X -0.042,Y -203.710,Z 837.859,A 0.000,B 0.000,C 90.000,E1 334.665} C_DIS
LIN {X 0.068,Y -209.253,Z 837.841,A 0.000,B 0.000,C 90.000,E1 331.435} C_DIS
LIN {X 0.027,Y -216.834,Z 837.820,A 0.000,B 0.000,C 90.000,E1 327.502} C_DIS
LIN {X -0.007,Y -223.517,Z 837.802,A 0.000,B 0.000,C 90.000,E1 324.402} C_DIS
LIN {X 0.017,Y -230.835,Z 837.785,A 0.000,B 0.000,C 90.000,E1 321.331} C_DIS
LIN {X -0.043,Y -239.938,Z 837.766,A 0.000,B 0.000,C 90.000,E1 317.957} C_DIS
LIN {X 0.133,Y -249.906,Z 837.748,A 0.000,B 0.000,C 90.000,E1 314.595} C_DIS
LIN {X -0.091,Y -260.826,Z 837.730,A 0.000,B 0.000,C 90.000,E1 311.391} C_DIS
LIN {X 0.045,Y -272.649,Z 837.712,A 0.000,B 0.000,C 90.000,E1 308.177} C_DIS
LIN {X -0.151,Y -285.431,Z 837.695,A 0.000,B 0.000,C 90.000,E1 305.105} C_DIS
LIN {X -0.079,Y -301.063,Z 837.676,A 0.000,B 0.000,C 90.000,E1 301.720} C_DIS
LIN {X 0.012,Y -314.860,Z 837.662,A 0.000,B 0.000,C 90.000,E1 299.077} C_DIS
LIN {X 0.072,Y -328.141,Z 837.649,A 0.000,B 0.000,C 90.000,E1 296.821} C_DIS
LIN {X 0.138,Y -348.825,Z 837.632,A 0.000,B 0.000,C 90.000,E1 293.695} C_DIS
LIN {X 0.081,Y -364.671,Z 837.620,A 0.000,B 0.000,C 90.000,E1 291.589} C_DIS
LIN {X -0.113,Y -381.775,Z 837.609,A 0.000,B 0.000,C 90.000,E1 289.577} C_DIS
LIN {X -0.113,Y -399.550,Z 837.598,A 0.000,B 0.000,C 90.000,E1 287.638} C_DIS
LIN {X -0.021,Y -412.432,Z 837.590,A 0.000,B 0.000,C 90.000,E1 286.260} C_DIS
LIN {X 0.084,Y -425.023,Z 837.583,A 0.000,B 0.000,C 90.000,E1 284.898} C_DIS
LIN {X -0.129,Y -437.264,Z 837.575,A 0.000,B 0.000,C 90.000,E1 283.592} C_DIS
LIN {X -0.148,Y -446.719,Z 837.570,A 0.000,B 0.000,C 90.000,E1 282.535} C_DIS
LIN {X -0.070,Y -455.600,Z 837.564,A 0.000,B 0.000,C 90.000,E1 281.478} C_DIS
LIN {X 0.027,Y -463.891,Z 837.558,A 0.000,B 0.000,C 90.000,E1 280.433} C_DIS
LIN {X -0.156,Y -471.594,Z 837.552,A 0.000,B 0.000,C 90.000,E1 279.434} C_DIS
LIN {X -0.202,Y -476.716,Z 837.548,A 0.000,B 0.000,C 90.000,E1 278.681} C_DIS
LIN {X 0.268,Y -481.245,Z 837.544,A 0.000,B 0.000,C 90.000,E1 277.871} C_DIS
LIN {X -0.050,Y -483.858,Z 837.541,A 0.000,B 0.000,C 90.000,E1 277.409} C_DIS
LIN {X 0.127,Y -486.096,Z 837.538,A 0.000,B 0.000,C 90.000,E1 276.891} C_DIS
LIN {X -0.164,Y -488.065,Z 837.536,A 0.000,B 0.000,C 90.000,E1 276.429} C_DIS
LIN {X 0.035,Y -489.729,Z 837.533,A 0.000,B 0.000,C 90.000,E1 275.910} C_DIS
LIN {X 0.246,Y -491.001,Z 837.530,A 0.000,B 0.000,C 90.000,E1 275.391} C_DIS
LIN {X -0.067,Y -491.942,Z 837.527,A 0.000,B 0.000,C 90.000,E1 274.935} C_DIS
LIN {X 0.162,Y -492.521,Z 837.525,A 0.000,B 0.000,C 90.000,E1 274.416} C_DIS
LIN {X -0.098,Y -492.687,Z 837.522,A 0.000,B 0.000,C 90.000,E1 273.955} C_DIS
LIN {X 0.104,Y -492.494,Z 837.519,A 0.000,B 0.000,C 90.000,E1 273.440} C_DIS
LIN {X -0.155,Y -491.996,Z 837.516,A 0.000,B 0.000,C 90.000,E1 272.980} C_DIS
LIN {X 0.050,Y -491.033,Z 837.514,A 0.000,B 0.000,C 90.000,E1 272.465} C_DIS
LIN {X -0.234,Y -489.612,Z 837.511,A 0.000,B 0.000,C 90.000,E1 272.007} C_DIS
LIN {X -0.020,Y -487.742,Z 837.508,A 0.000,B 0.000,C 90.000,E1 271.489} C_DIS
LIN {X 0.170,Y -485.350,Z 837.505,A 0.000,B 0.000,C 90.000,E1 270.974} C_DIS
LIN {X -0.140,Y -482.233,Z 837.503,A 0.000,B 0.000,C 90.000,E1 270.516} C_DIS
LIN {X 0.019,Y -478.569,Z 837.500,A 0.000,B 0.000,C 90.000,E1 270.000} C_DIS
LIN {X 0.156,Y -474.091,Z 837.497,A 0.000,B 0.000,C 90.000,E1 269.484} C_DIS
LIN {X -0.203,Y -468.584,Z 837.494,A 0.000,B 0.000,C 90.000,E1 269.026} C_DIS
LIN {X -0.167,Y -462.489,Z 837.492,A 0.000,B 0.000,C 90.000,E1 268.568} C_DIS
LIN {X -0.081,Y -455.812,Z 837.490,A 0.000,B 0.000,C 90.000,E1 268.165} C_DIS
LIN {X 0.081,Y -448.527,Z 837.488,A 0.000,B 0.000,C 90.000,E1 267.822} C_DIS
LIN {X -0.097,Y -440.980,Z 837.487,A 0.000,B 0.000,C 90.000,E1 267.593} C_DIS
LIN {X 0.167,Y -432.235,Z 837.485,A 0.000,B 0.000,C 90.000,E1 267.364} C_DIS
LIN {X 0.071,Y -422.856,Z 837.485,A 0.000,B 0.000,C 90.000,E1 267.249} C_DIS
LIN {X -0.084,Y -419.534,Z 837.485,A 0.000,B 0.000,C 90.000,E1 267.249} C_DIS
LIN {X -0.069,Y -181.017,Z 837.485,A 0.000,B 0.000,C 90.000,E1 267.249} C_DIS
LIN {X 0.063,Y -180.907,Z 837.475,A 0.000,B 0.000,C 90.000,E1 265.469} C_DIS
LIN {X -0.061,Y -180.745,Z 837.470,A 0.000,B 0.000,C 90.000,E1 264.666} C_DIS
LIN {X 0.008,Y -178.836,Z 837.442,A 0.000,B 0.000,C 90.000,E1 259.577} C_DIS
LIN {X -0.095,Y -175.881,Z 837.414,A 0.000,B 0.000,C 90.000,E1 254.519} C_DIS
LIN {X 0.012,Y -174.543,Z 837.404,A 0.000,B 0.000,C 90.000,E1 252.779} C_DIS
LIN {X 0.104,Y -171.527,Z 837.381,A 0.000,B 0.000,C 90.000,E1 248.465} C_DIS
LIN {X 0.089,Y -167.753,Z 837.357,A 0.000,B 0.000,C 90.000,E1 244.152} C_DIS
LIN {X 0.028,Y -166.457,Z 837.347,A 0.000,B 0.000,C 90.000,E1 242.436} C_DIS
LIN {X 0.017,Y -163.172,Z 837.328,A 0.000,B 0.000,C 90.000,E1 238.948} C_DIS
LIN {X 0.066,Y -161.132,Z 837.313,A 0.000,B 0.000,C 90.000,E1 236.294} C_DIS
LIN {X -0.031,Y -157.153,Z 837.288,A 0.000,B 0.000,C 90.000,E1 231.904} C_DIS
LIN {X -0.008,Y -155.886,Z 837.278,A 0.000,B 0.000,C 90.000,E1 230.114} C_DIS
LIN {X -0.049,Y -152.135,Z 837.253,A 0.000,B 0.000,C 90.000,E1 225.648} C_DIS
LIN {X -0.030,Y -150.385,Z 837.238,A 0.000,B 0.000,C 90.000,E1 222.933} C_DIS
LIN {X -0.005,Y -147.117,Z 837.213,A 0.000,B 0.000,C 90.000,E1 218.382} C_DIS
LIN {X -0.014,Y -145.682,Z 837.198,A 0.000,B 0.000,C 90.000,E1 215.644} C_DIS
LIN {X -0.015,Y -143.064,Z 837.172,A 0.000,B 0.000,C 90.000,E1 211.052} C_DIS
LIN {X 0.041,Y -141.686,Z 837.152,A 0.000,B 0.000,C 90.000,E1 207.334} C_DIS
LIN {X 0.020,Y -139.459,Z 837.116,A 0.000,B 0.000,C 90.000,E1 200.844} C_DIS
LIN {X 0.070,Y -139.193,Z 837.105,A 0.000,B 0.000,C 90.000,E1 198.960} C_DIS
LIN {X -0.043,Y -138.325,Z 837.054,A 0.000,B 0.000,C 90.000,E1 189.670} C_DIS
LIN {X -0.038,Y -139.453,Z 837.007,A 0.000,B 0.000,C 90.000,E1 181.260} C_DIS
LIN {X 0.042,Y -141.000,Z 836.976,A 0.000,B 0.000,C 90.000,E1 175.641} C_DIS
LIN {X -0.008,Y -142.755,Z 836.955,A 0.000,B 0.000,C 90.000,E1 171.951} C_DIS
LIN {X -0.053,Y -145.156,Z 836.930,A 0.000,B 0.000,C 90.000,E1 167.353} C_DIS
LIN {X -0.060,Y -147.779,Z 836.909,A 0.000,B 0.000,C 90.000,E1 163.685} C_DIS
LIN {X 0.020,Y -150.456,Z 836.889,A 0.000,B 0.000,C 90.000,E1 160.007} C_DIS
LIN {X -0.047,Y -153.905,Z 836.869,A 0.000,B 0.000,C 90.000,E1 156.410} C_DIS
LIN {X 0.019,Y -157.317,Z 836.849,A 0.000,B 0.000,C 90.000,E1 152.794} C_DIS
LIN {X -0.035,Y -161.504,Z 836.829,A 0.000,B 0.000,C 90.000,E1 149.253} C_DIS
LIN {X -0.020,Y -165.703,Z 836.810,A 0.000,B 0.000,C 90.000,E1 145.722} C_DIS
LIN {X 0.106,Y -170.648,Z 836.790,A 0.000,B 0.000,C 90.000,E1 142.190} C_DIS
LIN {X 0.020,Y -175.524,Z 836.771,A 0.000,B 0.000,C 90.000,E1 138.771} C_DIS
LIN {X 0.013,Y -181.143,Z 836.752,A 0.000,B 0.000,C 90.000,E1 135.364} C_DIS
LIN {X 0.011,Y -186.595,Z 836.733,A 0.000,B 0.000,C 90.000,E1 132.000} C_DIS
LIN {X 0.082,Y -191.206,Z 836.719,A 0.000,B 0.000,C 90.000,E1 129.483} C_DIS
LIN {X 0.108,Y -192.887,Z 836.714,A 0.000,B 0.000,C 90.000,E1 128.463} C_DIS
LIN {X 0.115,Y -293.974,Z 836.714,A 0.000,B 0.000,C 90.000,E1 128.463} C_DIS
LIN {X 0.099,Y -298.616,Z 836.713,A 0.000,B 0.000,C 90.000,E1 128.302} C_DIS
LIN {X -0.052,Y -300.796,Z 836.712,A 0.000,B 0.000,C 90.000,E1 128.177} C_DIS
LIN {X 0.014,Y -303.795,Z 836.710,A 0.000,B 0.000,C 90.000,E1 127.855} C_DIS
LIN {X -0.021,Y -307.419,Z 836.707,A 0.000,B 0.000,C 90.000,E1 127.282} C_DIS
LIN {X -0.002,Y -308.853,Z 836.705,A 0.000,B 0.000,C 90.000,E1 126.950} C_DIS
LIN {X -0.045,Y -309.978,Z 836.703,A 0.000,B 0.000,C 90.000,E1 126.629} C_DIS
LIN {X 0.073,Y -319.997,Z 836.685,A 0.000,B 0.000,C 90.000,E1 123.372} C_DIS
LIN {X -0.091,Y -330.322,Z 836.670,A 0.000,B 0.000,C 90.000,E1 120.541} C_DIS
LIN {X -0.009,Y -341.995,Z 836.654,A 0.000,B 0.000,C 90.000,E1 117.719} C_DIS
LIN {X 0.090,Y -355.112,Z 836.639,A 0.000,B 0.000,C 90.000,E1 114.951} C_DIS
LIN {X -0.117,Y -368.085,Z 836.625,A 0.000,B 0.000,C 90.000,E1 112.589} C_DIS
LIN {X -0.139,Y -382.386,Z 836.612,A 0.000,B 0.000,C 90.000,E1 110.248} C_DIS
LIN {X -0.065,Y -398.120,Z 836.600,A 0.000,B 0.000,C 90.000,E1 107.946} C_DIS
LIN {X -0.111,Y -415.397,Z 836.587,A 0.000,B 0.000,C 90.000,E1 105.717} C_DIS
LIN {X -0.065,Y -434.336,Z 836.575,A 0.000,B 0.000,C 90.000,E1 103.536} C_DIS
LIN {X 0.007,Y -454.397,Z 836.564,A 0.000,B 0.000,C 90.000,E1 101.478} C_DIS
LIN {X -0.203,Y -467.228,Z 836.557,A 0.000,B 0.000,C 90.000,E1 100.310} C_DIS
LIN {X -0.185,Y -469.385,Z 836.556,A 0.000,B 0.000,C 90.000,E1 100.074} C_DIS
LIN {X -0.249,Y -471.017,Z 836.555,A 0.000,B 0.000,C 90.000,E1 99.849} C_DIS
LIN {X 0.069,Y -472.365,Z 836.553,A 0.000,B 0.000,C 90.000,E1 99.557} C_DIS
LIN {X -0.079,Y -473.362,Z 836.552,A 0.000,B 0.000,C 90.000,E1 99.321} C_DIS
LIN {X 0.033,Y -474.499,Z 836.549,A 0.000,B 0.000,C 90.000,E1 98.803} C_DIS
LIN {X 0.223,Y -474.640,Z 836.546,A 0.000,B 0.000,C 90.000,E1 98.276} C_DIS
LIN {X -0.121,Y -473.810,Z 836.543,A 0.000,B 0.000,C 90.000,E1 97.814} C_DIS
LIN {X 0.007,Y -471.877,Z 836.541,A 0.000,B 0.000,C 90.000,E1 97.296} C_DIS
LIN {X 0.130,Y -468.702,Z 836.538,A 0.000,B 0.000,C 90.000,E1 96.777} C_DIS
LIN {X 0.185,Y -454.201,Z 836.525,A 0.000,B 0.000,C 90.000,E1 94.473} C_DIS
LIN {X -0.110,Y -443.604,Z 836.515,A 0.000,B 0.000,C 90.000,E1 92.694} C_DIS
LIN {X 0.082,Y -434.327,Z 836.506,A 0.000,B 0.000,C 90.000,E1 91.088} C_DIS
LIN {X -0.036,Y -426.370,Z 836.499,A 0.000,B 0.000,C 90.000,E1 89.771} C_DIS
LIN {X -0.039,Y -414.904,Z 836.488,A 0.000,B 0.000,C 90.000,E1 87.879} C_DIS
LIN {X 0.064,Y -405.054,Z 836.479,A 0.000,B 0.000,C 90.000,E1 86.216} C_DIS
LIN {X 0.090,Y -391.904,Z 836.467,A 0.000,B 0.000,C 90.000,E1 83.976} C_DIS
LIN {X -0.110,Y -379.032,Z 836.454,A 0.000,B 0.000,C 90.000,E1 81.724} C_DIS
LIN {X -0.136,Y -364.907,Z 836.439,A 0.000,B 0.000,C 90.000,E1 79.106} C_DIS
LIN {X 0.019,Y -352.856,Z 836.426,A 0.000,B 0.000,C 90.000,E1 76.700} C_DIS
LIN {X 0.046,Y -342.421,Z 836.414,A 0.000,B 0.000,C 90.000,E1 74.574} C_DIS
LIN {X -0.092,Y -330.531,Z 836.401,A 0.000,B 0.000,C 90.000,E1 72.127} C_DIS
LIN {X 0.100,Y -318.925,Z 836.387,A 0.000,B 0.000,C 90.000,E1 69.571} C_DIS
LIN {X -0.056,Y -303.526,Z 836.367,A 0.000,B 0.000,C 90.000,E1 66.049} C_DIS
LIN {X 0.058,Y -291.517,Z 836.350,A 0.000,B 0.000,C 90.000,E1 63.050} C_DIS
LIN {X 0.135,Y -281.211,Z 836.335,A 0.000,B 0.000,C 90.000,E1 60.333} C_DIS
LIN {X 0.058,Y -270.036,Z 836.318,A 0.000,B 0.000,C 90.000,E1 57.248} C_DIS
LIN {X -0.050,Y -258.399,Z 836.299,A 0.000,B 0.000,C 90.000,E1 53.749} C_DIS
LIN {X -0.062,Y -248.515,Z 836.281,A 0.000,B 0.000,C 90.000,E1 50.517} C_DIS
LIN {X 0.066,Y -238.210,Z 836.260,A 0.000,B 0.000,C 90.000,E1 46.824} C_DIS
LIN {X 0.024,Y -228.740,Z 836.239,A 0.000,B 0.000,C 90.000,E1 43.095} C_DIS
LIN {X -0.133,Y -221.535,Z 836.223,A 0.000,B 0.000,C 90.000,E1 40.092} C_DIS
LIN {X 0.066,Y -212.994,Z 836.201,A 0.000,B 0.000,C 90.000,E1 36.171} C_DIS
LIN {X -0.037,Y -205.162,Z 836.179,A 0.000,B 0.000,C 90.000,E1 32.260} C_DIS
LIN {X -0.089,Y -199.439,Z 836.161,A 0.000,B 0.000,C 90.000,E1 29.077} C_DIS
LIN {X 0.055,Y -194.417,Z 836.143,A 0.000,B 0.000,C 90.000,E1 25.796} C_DIS
LIN {X 0.081,Y -190.200,Z 836.125,A 0.000,B 0.000,C 90.000,E1 22.514} C_DIS
LIN {X -0.043,Y -186.039,Z 836.102,A 0.000,B 0.000,C 90.000,E1 18.417} C_DIS
LIN {X -0.042,Y -183.011,Z 836.079,A 0.000,B 0.000,C 90.000,E1 14.245} C_DIS
LIN {X -0.077,Y -180.453,Z 836.042,A 0.000,B 0.000,C 90.000,E1 7.530} C_DIS
LIN {X -0.003,Y -181.783,Z 835.979,A 0.000,B 0.000,C 90.000,E1 356.159} C_DIS
LIN {X -0.071,Y -184.747,Z 835.951,A 0.000,B 0.000,C 90.000,E1 351.141} C_DIS
LIN {X 0.034,Y -188.234,Z 835.927,A 0.000,B 0.000,C 90.000,E1 346.937} C_DIS
LIN {X 0.103,Y -192.621,Z 835.904,A 0.000,B 0.000,C 90.000,E1 342.779} C_DIS
LIN {X -0.017,Y -197.868,Z 835.882,A 0.000,B 0.000,C 90.000,E1 338.720} C_DIS
LIN {X 0.015,Y -203.936,Z 835.859,A 0.000,B 0.000,C 90.000,E1 334.665} C_DIS
LIN {X 0.032,Y -209.460,Z 835.841,A 0.000,B 0.000,C 90.000,E1 331.463} C_DIS
LIN {X -0.016,Y -217.045,Z 835.820,A 0.000,B 0.000,C 90.000,E1 327.533} C_DIS
LIN {X 0.074,Y -223.722,Z 835.802,A 0.000,B 0.000,C 90.000,E1 324.402} C_DIS
LIN {X -0.075,Y -231.038,Z 835.785,A 0.000,B 0.000,C 90.000,E1 321.376} C_DIS
LIN {X 0.057,Y -240.144,Z 835.766,A 0.000,B 0.000,C 90.000,E1 317.957} C_DIS
LIN {X -0.113,Y -250.072,Z 835.748,A 0.000,B 0.000,C 90.000,E1 314.676} C_DIS
LIN {X 0.027,Y -260.962,Z 835.730,A 0.000,B 0.000,C 90.000,E1 311.391} C_DIS
LIN {X -0.043,Y -272.739,Z 835.712,A 0.000,B 0.000,C 90.000,E1 308.222} C_DIS
LIN {X -0.016,Y -285.450,Z 835.695,A 0.000,B 0.000,C 90.000,E1 305.105} C_DIS
LIN {X 0.062,Y -301.008,Z 835.676,A 0.000,B 0.000,C 90.000,E1 301.720} C_DIS
LIN {X 0.060,Y -316.576,Z 835.660,A 0.000,B 0.000,C 90.000,E1 298.771} C_DIS
LIN {X -0.022,Y -331.987,Z 835.646,A 0.000,B 0.000,C 90.000,E1 296.232} C_DIS
LIN {X 0.010,Y -352.962,Z 835.629,A 0.000,B 0.000,C 90.000,E1 293.131} C_DIS
LIN {X -0.097,Y -369.160,Z 835.617,A 0.000,B 0.000,C 90.000,E1 291.046} C_DIS
LIN {X -0.037,Y -389.184,Z 835.604,A 0.000,B 0.000,C 90.000,E1 288.725} C_DIS
LIN {X 0.051,Y -404.735,Z 835.595,A 0.000,B 0.000,C 90.000,E1 287.040} C_DIS
LIN {X -0.071,Y -414.981,Z 835.589,A 0.000,B 0.000,C 90.000,E1 285.969} C_DIS
LIN {X 0.126,Y -427.612,Z 835.581,A 0.000,B 0.000,C 90.000,E1 284.592} C_DIS
LIN {X -0.202,Y -439.771,Z 835.574,A 0.000,B 0.000,C 90.000,E1 283.300} C_DIS
LIN {X -0.207,Y -449.099,Z 835.568,A 0.000,B 0.000,C 90.000,E1 282.243} C_DIS
LIN {X -0.102,Y -457.821,Z 835.562,A 0.000,B 0.000,C 90.000,E1 281.186} C_DIS
LIN {X 0.022,Y -466.018,Z 835.556,A 0.000,B 0.000,C 90.000,E1 280.141} C_DIS
LIN {X 0.006,Y -471.714,Z 835.552,A 0.000,B 0.000,C 90.000,E1 279.378} C_DIS
LIN {X -0.035,Y -476.821,Z 835.548,A 0.000,B 0.000,C 90.000,E1 278.624} C_DIS
LIN {X -0.038,Y -481.306,Z 835.544,A 0.000,B 0.000,C 90.000,E1 277.871} C_DIS
LIN {X -0.059,Y -485.054,Z 835.540,A 0.000,B 0.000,C 90.000,E1 277.125} C_DIS
LIN {X 0.011,Y -488.124,Z 835.535,A 0.000,B 0.000,C 90.000,E1 276.372} C_DIS
LIN {X 0.212,Y -489.764,Z 835.533,A 0.000,B 0.000,C 90.000,E1 275.853} C_DIS
LIN {X -0.065,Y -491.038,Z 835.530,A 0.000,B 0.000,C 90.000,E1 275.391} C_DIS
LIN {X 0.113,Y -491.960,Z 835.527,A 0.000,B 0.000,C 90.000,E1 274.878} C_DIS
LIN {X -0.149,Y -492.522,Z 835.524,A 0.000,B 0.000,C 90.000,E1 274.416} C_DIS
LIN {X 0.083,Y -492.691,Z 835.522,A 0.000,B 0.000,C 90.000,E1 273.898} C_DIS
LIN {X -0.207,Y -492.503,Z 835.519,A 0.000,B 0.000,C 90.000,E1 273.440} C_DIS
LIN {X 0.026,Y -491.973,Z 835.516,A 0.000,B 0.000,C 90.000,E1 272.922} C_DIS
LIN {X 0.231,Y -491.001,Z 835.514,A 0.000,B 0.000,C 90.000,E1 272.407} C_DIS
LIN {X -0.055,Y -489.572,Z 835.511,A 0.000,B 0.000,C 90.000,E1 271.949} C_DIS
LIN {X 0.159,Y -487.660,Z 835.508,A 0.000,B 0.000,C 90.000,E1 271.432} C_DIS
LIN {X -0.136,Y -485.272,Z 835.505,A 0.000,B 0.000,C 90.000,E1 270.974} C_DIS
LIN {X 0.037,Y -482.244,Z 835.503,A 0.000,B 0.000,C 90.000,E1 270.458} C_DIS
LIN {X 0.194,Y -478.500,Z 835.500,A 0.000,B 0.000,C 90.000,E1 269.943} C_DIS
LIN {X -0.145,Y -473.926,Z 835.497,A 0.000,B 0.000,C 90.000,E1 269.484} C_DIS
LIN {X -0.032,Y -468.452,Z 835.494,A 0.000,B 0.000,C 90.000,E1 268.969} C_DIS
LIN {X -0.001,Y -462.320,Z 835.492,A 0.000,B 0.000,C 90.000,E1 268.511} C_DIS
LIN {X 0.100,Y -455.664,Z 835.490,A 0.000,B 0.000,C 90.000,E1 268.108} C_DIS
LIN {X 0.175,Y -452.257,Z 835.489,A 0.000,B 0.000,C 90.000,E1 267.936} C_DIS
LIN {X 0.179,Y -444.819,Z 835.487,A 0.000,B 0.000,C 90.000,E1 267.650} C_DIS
LIN {X -0.192,Y -436.934,Z 835.486,A 0.000,B 0.000,C 90.000,E1 267.478} C_DIS
LIN {X -0.105,Y -428.021,Z 835.485,A 0.000,B 0.000,C 90.000,E1 267.306} C_DIS
LIN {X 0.114,Y -418.474,Z 835.484,A 0.000,B 0.000,C 90.000,E1 267.192} C_DIS
LIN {X 0.017,Y -181.014,Z 835.484,A 0.000,B 0.000,C 90.000,E1 267.192} C_DIS
LIN {X -0.027,Y -180.906,Z 835.475,A 0.000,B 0.000,C 90.000,E1 265.469} C_DIS
LIN {X 0.030,Y -180.733,Z 835.470,A 0.000,B 0.000,C 90.000,E1 264.609} C_DIS
LIN {X -0.049,Y -178.822,Z 835.442,A 0.000,B 0.000,C 90.000,E1 259.567} C_DIS
LIN {X 0.034,Y -175.867,Z 835.414,A 0.000,B 0.000,C 90.000,E1 254.448} C_DIS
LIN {X 0.028,Y -173.836,Z 835.399,A 0.000,B 0.000,C 90.000,E1 251.891} C_DIS
LIN {X 0.017,Y -171.503,Z 835.380,A 0.000,B 0.000,C 90.000,E1 248.465} C_DIS
LIN {X 0.003,Y -167.731,Z 835.356,A 0.000,B 0.000,C 90.000,E1 244.152} C_DIS
LIN {X 0.020,Y -166.428,Z 835.347,A 0.000,B 0.000,C 90.000,E1 242.410} C_DIS
LIN {X 0.017,Y -163.148,Z 835.327,A 0.000,B 0.000,C 90.000,E1 238.918} C_DIS
LIN {X -0.017,Y -161.104,Z 835.313,A 0.000,B 0.000,C 90.000,E1 236.294} C_DIS
LIN {X -0.034,Y -157.830,Z 835.293,A 0.000,B 0.000,C 90.000,E1 232.763} C_DIS
LIN {X 0.029,Y -155.863,Z 835.278,A 0.000,B 0.000,C 90.000,E1 230.070} C_DIS
LIN {X 0.085,Y -152.114,Z 835.253,A 0.000,B 0.000,C 90.000,E1 225.567} C_DIS
LIN {X -0.007,Y -150.364,Z 835.238,A 0.000,B 0.000,C 90.000,E1 222.894} C_DIS
LIN {X 0.031,Y -147.099,Z 835.213,A 0.000,B 0.000,C 90.000,E1 218.338} C_DIS
LIN {X 0.026,Y -145.668,Z 835.198,A 0.000,B 0.000,C 90.000,E1 215.598} C_DIS
LIN {X 0.029,Y -143.050,Z 835.172,A 0.000,B 0.000,C 90.000,E1 211.003} C_DIS
LIN {X -0.036,Y -141.673,Z 835.152,A 0.000,B 0.000,C 90.000,E1 207.334} C_DIS
LIN {X 0.073,Y -139.454,Z 835.116,A 0.000,B 0.000,C 90.000,E1 200.791} C_DIS
LIN {X -0.006,Y -139.188,Z 835.105,A 0.000,B 0.000,C 90.000,E1 198.960} C_DIS
LIN {X 0.017,Y -138.322,Z 835.053,A 0.000,B 0.000,C 90.000,E1 189.613} C_DIS
LIN {X 0.024,Y -139.459,Z 835.007,A 0.000,B 0.000,C 90.000,E1 181.203} C_DIS
LIN {X -0.035,Y -141.013,Z 834.976,A 0.000,B 0.000,C 90.000,E1 175.641} C_DIS
LIN {X 0.055,Y -142.767,Z 834.955,A 0.000,B 0.000,C 90.000,E1 171.894} C_DIS
LIN {X 0.010,Y -145.176,Z 834.929,A 0.000,B 0.000,C 90.000,E1 167.297} C_DIS
LIN {X 0.043,Y -147.798,Z 834.909,A 0.000,B 0.000,C 90.000,E1 163.614} C_DIS
LIN {X -0.061,Y -150.482,Z 834.889,A 0.000,B 0.000,C 90.000,E1 160.007} C_DIS
LIN {X 0.012,Y -153.937,Z 834.869,A 0.000,B 0.000,C 90.000,E1 156.357} C_DIS
LIN {X 0.076,Y -157.348,Z 834.849,A 0.000,B 0.000,C 90.000,E1 152.743} C_DIS
LIN {X 0.019,Y -161.542,Z 834.829,A 0.000,B 0.000,C 90.000,E1 149.203} C_DIS
LIN {X 0.032,Y -165.740,Z 834.809,A 0.000,B 0.000,C 90.000,E1 145.674} C_DIS
LIN {X 0.019,Y -170.693,Z 834.790,A 0.000,B 0.000,C 90.000,E1 142.190} C_DIS
LIN {X -0.070,Y -175.568,Z 834.771,A 0.000,B 0.000,C 90.000,E1 138.771} C_DIS
LIN {X 0.050,Y -181.186,Z 834.752,A 0.000,B 0.000,C 90.000,E1 135.324} C_DIS
LIN {X -0.081,Y -186.646,Z 834.733,A 0.000,B 0.000,C 90.000,E1 132.000} C_DIS
LIN {X -0.012,Y -191.251,Z 834.719,A 0.000,B 0.000,C 90.000,E1 129.483} C_DIS
LIN {X -0.023,Y -192.876,Z 834.714,A 0.000,B 0.000,C 90.000,E1 128.508} C_DIS
LIN {X 0.160,Y -293.786,Z 834.714,A 0.000,B 0.000,C 90.000,E1 128.463} C_DIS
LIN {X -0.078,Y -295.928,Z 834.714,A 0.000,B 0.000,C 90.000,E1 128.463} C_DIS
LIN {X -0.012,Y -301.161,Z 834.712,A 0.000,B 0.000,C 90.000,E1 128.141} C_DIS
LIN {X 0.107,Y -304.029,Z 834.710,A 0.000,B 0.000,C 90.000,E1 127.810} C_DIS
LIN {X 0.038,Y -306.057,Z 834.708,A 0.000,B 0.000,C 90.000,E1 127.523} C_DIS
LIN {X -0.033,Y -307.642,Z 834.707,A 0.000,B 0.000,C 90.000,E1 127.237} C_DIS
LIN {X 0.181,Y -309.014,Z 834.705,A 0.000,B 0.000,C 90.000,E1 126.870} C_DIS
LIN {X -0.030,Y -311.979,Z 834.700,A 0.000,B 0.000,C 90.000,E1 125.931} C_DIS
LIN {X -0.017,Y -322.313,Z 834.682,A 0.000,B 0.000,C 90.000,E1 122.704} C_DIS
LIN {X -0.114,Y -332.949,Z 834.666,A 0.000,B 0.000,C 90.000,E1 119.873} C_DIS
LIN {X 0.036,Y -344.956,Z 834.650,A 0.000,B 0.000,C 90.000,E1 117.052} C_DIS
LIN {X -0.090,Y -358.434,Z 834.635,A 0.000,B 0.000,C 90.000,E1 114.335} C_DIS
LIN {X -0.076,Y -371.751,Z 834.622,A 0.000,B 0.000,C 90.000,E1 111.950} C_DIS
LIN {X -0.150,Y -386.426,Z 834.609,A 0.000,B 0.000,C 90.000,E1 109.631} C_DIS
LIN {X 0.019,Y -402.559,Z 834.596,A 0.000,B 0.000,C 90.000,E1 107.330} C_DIS
LIN {X -0.151,Y -420.271,Z 834.584,A 0.000,B 0.000,C 90.000,E1 105.134} C_DIS
LIN {X 0.177,Y -439.618,Z 834.572,A 0.000,B 0.000,C 90.000,E1 102.939} C_DIS
LIN {X 0.082,Y -459.833,Z 834.561,A 0.000,B 0.000,C 90.000,E1 100.950} C_DIS
LIN {X -0.011,Y -467.545,Z 834.557,A 0.000,B 0.000,C 90.000,E1 100.254} C_DIS
LIN {X 0.002,Y -469.630,Z 834.556,A 0.000,B 0.000,C 90.000,E1 100.018} C_DIS
LIN {X -0.067,Y -471.212,Z 834.554,A 0.000,B 0.000,C 90.000,E1 99.792} C_DIS
LIN {X -0.213,Y -472.512,Z 834.553,A 0.000,B 0.000,C 90.000,E1 99.557} C_DIS
LIN {X 0.107,Y -473.472,Z 834.552,A 0.000,B 0.000,C 90.000,E1 99.265} C_DIS
LIN {X -0.248,Y -474.545,Z 834.549,A 0.000,B 0.000,C 90.000,E1 98.803} C_DIS
LIN {X -0.058,Y -474.628,Z 834.546,A 0.000,B 0.000,C 90.000,E1 98.276} C_DIS
LIN {X 0.069,Y -473.738,Z 834.543,A 0.000,B 0.000,C 90.000,E1 97.757} C_DIS
LIN {X 0.197,Y -471.729,Z 834.540,A 0.000,B 0.000,C 90.000,E1 97.239} C_DIS
LIN {X -0.043,Y -465.197,Z 834.535,A 0.000,B 0.000,C 90.000,E1 96.258} C_DIS
LIN {X -0.075,Y -450.993,Z 834.522,A 0.000,B 0.000,C 90.000,E1 93.955} C_DIS
LIN {X -0.195,Y -441.893,Z 834.513,A 0.000,B 0.000,C 90.000,E1 92.407} C_DIS
LIN {X -0.029,Y -432.583,Z 834.504,A 0.000,B 0.000,C 90.000,E1 90.802} C_DIS
LIN {X -0.039,Y -422.920,Z 834.496,A 0.000,B 0.000,C 90.000,E1 89.198} C_DIS
LIN {X -0.114,Y -411.480,Z 834.485,A 0.000,B 0.000,C 90.000,E1 87.306} C_DIS
LIN {X -0.049,Y -401.570,Z 834.476,A 0.000,B 0.000,C 90.000,E1 85.641} C_DIS
LIN {X -0.056,Y -386.875,Z 834.462,A 0.000,B 0.000,C 90.000,E1 83.109} C_DIS
LIN {X 0.061,Y -374.092,Z 834.449,A 0.000,B 0.000,C 90.000,E1 80.792} C_DIS
LIN {X -0.161,Y -357.217,Z 834.431,A 0.000,B 0.000,C 90.000,E1 77.589} C_DIS
LIN {X -0.117,Y -345.286,Z 834.418,A 0.000,B 0.000,C 90.000,E1 75.172} C_DIS
LIN {X -0.072,Y -334.841,Z 834.406,A 0.000,B 0.000,C 90.000,E1 73.015} C_DIS
LIN {X 0.021,Y -323.174,Z 834.392,A 0.000,B 0.000,C 90.000,E1 70.496} C_DIS
LIN {X 0.057,Y -310.300,Z 834.376,A 0.000,B 0.000,C 90.000,E1 67.614} C_DIS
LIN {X -0.062,Y -299.438,Z 834.361,A 0.000,B 0.000,C 90.000,E1 65.025} C_DIS
LIN {X -0.042,Y -288.942,Z 834.346,A 0.000,B 0.000,C 90.000,E1 62.359} C_DIS
LIN {X -0.139,Y -278.759,Z 834.331,A 0.000,B 0.000,C 90.000,E1 59.665} C_DIS
LIN {X 0.023,Y -266.640,Z 834.312,A 0.000,B 0.000,C 90.000,E1 56.167} C_DIS
LIN {X 0.070,Y -256.368,Z 834.294,A 0.000,B 0.000,C 90.000,E1 52.970} C_DIS
LIN {X -0.034,Y -246.624,Z 834.276,A 0.000,B 0.000,C 90.000,E1 49.747} C_DIS
LIN {X 0.036,Y -236.491,Z 834.256,A 0.000,B 0.000,C 90.000,E1 46.053} C_DIS
LIN {X 0.100,Y -227.163,Z 834.235,A 0.000,B 0.000,C 90.000,E1 42.285} C_DIS
LIN {X -0.078,Y -220.035,Z 834.218,A 0.000,B 0.000,C 90.000,E1 39.277} C_DIS
LIN {X -0.055,Y -211.624,Z 834.197,A 0.000,B 0.000,C 90.000,E1 35.391} C_DIS
LIN {X 0.036,Y -203.936,Z 834.175,A 0.000,B 0.000,C 90.000,E1 31.416} C_DIS
LIN {X -0.041,Y -198.391,Z 834.157,A 0.000,B 0.000,C 90.000,E1 28.231} C_DIS
LIN {X 0.074,Y -193.559,Z 834.139,A 0.000,B 0.000,C 90.000,E1 24.951} C_DIS
LIN {X -0.078,Y -189.556,Z 834.121,A 0.000,B 0.000,C 90.000,E1 21.716} C_DIS
LIN {X -0.099,Y -185.632,Z 834.098,A 0.000,B 0.000,C 90.000,E1 17.583} C_DIS
LIN {X 0.013,Y -182.411,Z 834.070,A 0.000,B 0.000,C 90.000,E1 12.535} C_DIS
LIN {X -0.035,Y -180.418,Z 834.023,A 0.000,B 0.000,C 90.000,E1 4.131} C_DIS
LIN {X 0.005,Y -182.105,Z 833.979,A 0.000,B 0.000,C 90.000,E1 356.159} C_DIS
LIN {X -0.052,Y -185.044,Z 833.951,A 0.000,B 0.000,C 90.000,E1 351.141} C_DIS
LIN {X 0.063,Y -188.517,Z 833.928,A 0.000,B 0.000,C 90.000,E1 346.937} C_DIS
LIN {X -0.043,Y -192.874,Z 833.905,A 0.000,B 0.000,C 90.000,E1 342.834} C_DIS
LIN {X 0.031,Y -198.113,Z 833.882,A 0.000,B 0.000,C 90.000,E1 338.720} C_DIS
LIN {X 0.072,Y -204.164,Z 833.859,A 0.000,B 0.000,C 90.000,E1 334.665} C_DIS
LIN {X -0.088,Y -209.665,Z 833.842,A 0.000,B 0.000,C 90.000,E1 331.513} C_DIS
LIN {X 0.057,Y -217.259,Z 833.820,A 0.000,B 0.000,C 90.000,E1 327.533} C_DIS
LIN {X 0.024,Y -223.929,Z 833.802,A 0.000,B 0.000,C 90.000,E1 324.436} C_DIS
LIN {X 0.014,Y -231.242,Z 833.785,A 0.000,B 0.000,C 90.000,E1 321.376} C_DIS
LIN {X -0.024,Y -240.344,Z 833.767,A 0.000,B 0.000,C 90.000,E1 318.000} C_DIS
LIN {X -0.006,Y -250.225,Z 833.748,A 0.000,B 0.000,C 90.000,E1 314.676} C_DIS
LIN {X -0.052,Y -261.079,Z 833.730,A 0.000,B 0.000,C 90.000,E1 311.434} C_DIS
LIN {X -0.087,Y -272.810,Z 833.712,A 0.000,B 0.000,C 90.000,E1 308.257} C_DIS
LIN {X 0.116,Y -285.469,Z 833.695,A 0.000,B 0.000,C 90.000,E1 305.105} C_DIS
LIN {X 0.044,Y -300.957,Z 833.676,A 0.000,B 0.000,C 90.000,E1 301.750} C_DIS
LIN {X -0.073,Y -316.480,Z 833.660,A 0.000,B 0.000,C 90.000,E1 298.821} C_DIS
LIN {X 0.029,Y -329.854,Z 833.648,A 0.000,B 0.000,C 90.000,E1 296.565} C_DIS
LIN {X 0.003,Y -350.519,Z 833.630,A 0.000,B 0.000,C 90.000,E1 293.462} C_DIS
LIN {X 0.058,Y -368.866,Z 833.617,A 0.000,B 0.000,C 90.000,E1 291.046} C_DIS
LIN {X 0.018,Y -388.915,Z 833.604,A 0.000,B 0.000,C 90.000,E1 288.725} C_DIS
LIN {X 0.098,Y -404.471,Z 833.595,A 0.000,B 0.000,C 90.000,E1 287.040} C_DIS
LIN {X -0.143,Y -417.189,Z 833.587,A 0.000,B 0.000,C 90.000,E1 285.717} C_DIS
LIN {X -0.055,Y -429.762,Z 833.580,A 0.000,B 0.000,C 90.000,E1 284.356} C_DIS
LIN {X 0.061,Y -441.879,Z 833.572,A 0.000,B 0.000,C 90.000,E1 283.008} C_DIS
LIN {X 0.087,Y -451.086,Z 833.566,A 0.000,B 0.000,C 90.000,E1 281.951} C_DIS
LIN {X 0.221,Y -459.703,Z 833.561,A 0.000,B 0.000,C 90.000,E1 280.894} C_DIS
LIN {X -0.087,Y -467.754,Z 833.555,A 0.000,B 0.000,C 90.000,E1 279.905} C_DIS
LIN {X -0.162,Y -473.250,Z 833.551,A 0.000,B 0.000,C 90.000,E1 279.151} C_DIS
LIN {X -0.193,Y -478.191,Z 833.547,A 0.000,B 0.000,C 90.000,E1 278.398} C_DIS
LIN {X -0.176,Y -482.473,Z 833.542,A 0.000,B 0.000,C 90.000,E1 277.644} C_DIS
LIN {X -0.129,Y -486.028,Z 833.538,A 0.000,B 0.000,C 90.000,E1 276.891} C_DIS
LIN {X 0.063,Y -488.038,Z 833.535,A 0.000,B 0.000,C 90.000,E1 276.372} C_DIS
LIN {X -0.224,Y -489.677,Z 833.533,A 0.000,B 0.000,C 90.000,E1 275.910} C_DIS
LIN {X -0.014,Y -490.967,Z 833.530,A 0.000,B 0.000,C 90.000,E1 275.391} C_DIS
LIN {X 0.163,Y -491.904,Z 833.527,A 0.000,B 0.000,C 90.000,E1 274.878} C_DIS
LIN {X -0.099,Y -492.487,Z 833.524,A 0.000,B 0.000,C 90.000,E1 274.416} C_DIS
LIN {X 0.132,Y -492.701,Z 833.522,A 0.000,B 0.000,C 90.000,E1 273.898} C_DIS
LIN {X -0.157,Y -492.521,Z 833.519,A 0.000,B 0.000,C 90.000,E1 273.440} C_DIS
LIN {X 0.075,Y -491.998,Z 833.516,A 0.000,B 0.000,C 90.000,E1 272.922} C_DIS
LIN {X -0.210,Y -491.072,Z 833.514,A 0.000,B 0.000,C 90.000,E1 272.465} C_DIS
LIN {X -0.005,Y -489.672,Z 833.511,A 0.000,B 0.000,C 90.000,E1 271.949} C_DIS
LIN {X 0.210,Y -487.813,Z 833.508,A 0.000,B 0.000,C 90.000,E1 271.432} C_DIS
LIN {X -0.087,Y -485.398,Z 833.505,A 0.000,B 0.000,C 90.000,E1 270.974} C_DIS
LIN {X 0.088,Y -482.433,Z 833.503,A 0.000,B 0.000,C 90.000,E1 270.458} C_DIS
LIN {X -0.234,Y -478.773,Z 833.500,A 0.000,B 0.000,C 90.000,E1 270.000} C_DIS
LIN {X -0.094,Y -474.271,Z 833.497,A 0.000,B 0.000,C 90.000,E1 269.484} C_DIS
LIN {X 0.020,Y -468.848,Z 833.494,A 0.000,B 0.000,C 90.000,E1 268.969} C_DIS
LIN {X 0.023,Y -462.702,Z 833.492,A 0.000,B 0.000,C 90.000,E1 268.511} C_DIS
LIN {X -0.175,Y -459.713,Z 833.491,A 0.000,B 0.000,C 90.000,E1 268.339} C_DIS
LIN {X 0.182,Y -452.813,Z 833.489,A 0.000,B 0.000,C 90.000,E1 267.936} C_DIS
LIN {X 0.143,Y -445.451,Z 833.487,A 0.000,B 0.000,C 90.000,E1 267.650} C_DIS
LIN {X 0.149,Y -437.509,Z 833.486,A 0.000,B 0.000,C 90.000,E1 267.421} C_DIS
LIN {X 0.207,Y -428.753,Z 833.485,A 0.000,B 0.000,C 90.000,E1 267.249} C_DIS
LIN {X -0.010,Y -419.835,Z 833.484,A 0.000,B 0.000,C 90.000,E1 267.192} C_DIS
LIN {X -0.037,Y -181.011,Z 833.484,A 0.000,B 0.000,C 90.000,E1 267.192} C_DIS
LIN {X -0.085,Y -180.906,Z 833.475,A 0.000,B 0.000,C 90.000,E1 265.469} C_DIS
LIN {X -0.028,Y -180.724,Z 833.470,A 0.000,B 0.000,C 90.000,E1 264.609} C_DIS
LIN {X 0.070,Y -178.813,Z 833.442,A 0.000,B 0.000,C 90.000,E1 259.511} C_DIS
LIN {X -0.024,Y -175.858,Z 833.414,A 0.000,B 0.000,C 90.000,E1 254.448} C_DIS
LIN {X -0.042,Y -173.186,Z 833.395,A 0.000,B 0.000,C 90.000,E1 251.040} C_DIS
LIN {X -0.040,Y -171.488,Z 833.380,A 0.000,B 0.000,C 90.000,E1 248.465} C_DIS
LIN {X -0.052,Y -167.717,Z 833.356,A 0.000,B 0.000,C 90.000,E1 244.152} C_DIS
LIN {X -0.036,Y -166.408,Z 833.347,A 0.000,B 0.000,C 90.000,E1 242.410} C_DIS
LIN {X -0.038,Y -163.132,Z 833.327,A 0.000,B 0.000,C 90.000,E1 238.918} C_DIS
LIN {X -0.071,Y -161.084,Z 833.313,A 0.000,B 0.000,C 90.000,E1 236.294} C_DIS
LIN {X 0.039,Y -157.814,Z 833.293,A 0.000,B 0.000,C 90.000,E1 232.718} C_DIS
LIN {X -0.024,Y -155.849,Z 833.278,A 0.000,B 0.000,C 90.000,E1 230.070} C_DIS
LIN {X 0.033,Y -152.099,Z 833.253,A 0.000,B 0.000,C 90.000,E1 225.567} C_DIS
LIN {X 0.051,Y -150.350,Z 833.238,A 0.000,B 0.000,C 90.000,E1 222.852} C_DIS
LIN {X -0.020,Y -147.087,Z 833.213,A 0.000,B 0.000,C 90.000,E1 218.338} C_DIS
LIN {X -0.025,Y -145.658,Z 833.198,A 0.000,B 0.000,C 90.000,E1 215.598} C_DIS
LIN {X -0.021,Y -143.041,Z 833.172,A 0.000,B 0.000,C 90.000,E1 211.003} C_DIS
LIN {X -0.021,Y -141.665,Z 833.152,A 0.000,B 0.000,C 90.000,E1 207.308} C_DIS
LIN {X 0.024,Y -139.450,Z 833.116,A 0.000,B 0.000,C 90.000,E1 200.791} C_DIS
LIN {X -0.055,Y -139.184,Z 833.105,A 0.000,B 0.000,C 90.000,E1 198.960} C_DIS
LIN {X -0.032,Y -138.321,Z 833.053,A 0.000,B 0.000,C 90.000,E1 189.613} C_DIS
LIN {X -0.025,Y -139.462,Z 833.007,A 0.000,B 0.000,C 90.000,E1 181.203} C_DIS
LIN {X 0.055,Y -141.021,Z 832.976,A 0.000,B 0.000,C 90.000,E1 175.584} C_DIS
LIN {X 0.010,Y -142.386,Z 832.960,A 0.000,B 0.000,C 90.000,E1 172.818} C_DIS
LIN {X -0.069,Y -144.616,Z 832.934,A 0.000,B 0.000,C 90.000,E1 168.229} C_DIS
LIN {X -0.008,Y -147.811,Z 832.909,A 0.000,B 0.000,C 90.000,E1 163.614} C_DIS
LIN {X 0.079,Y -150.499,Z 832.889,A 0.000,B 0.000,C 90.000,E1 159.934} C_DIS
LIN {X -0.040,Y -153.956,Z 832.869,A 0.000,B 0.000,C 90.000,E1 156.357} C_DIS
LIN {X 0.022,Y -157.369,Z 832.849,A 0.000,B 0.000,C 90.000,E1 152.743} C_DIS
LIN {X -0.035,Y -161.568,Z 832.829,A 0.000,B 0.000,C 90.000,E1 149.203} C_DIS
LIN {X -0.023,Y -165.766,Z 832.809,A 0.000,B 0.000,C 90.000,E1 145.674} C_DIS
LIN {X -0.038,Y -170.723,Z 832.790,A 0.000,B 0.000,C 90.000,E1 142.190} C_DIS
LIN {X 0.005,Y -175.596,Z 832.771,A 0.000,B 0.000,C 90.000,E1 138.728} C_DIS
LIN {X -0.008,Y -181.213,Z 832.752,A 0.000,B 0.000,C 90.000,E1 135.324} C_DIS
LIN {X -0.016,Y -186.678,Z 832.733,A 0.000,B 0.000,C 90.000,E1 131.962} C_DIS
LIN {X -0.073,Y -191.280,Z 832.719,A 0.000,B 0.000,C 90.000,E1 129.483} C_DIS
LIN {X -0.088,Y -192.849,Z 832.714,A 0.000,B 0.000,C 90.000,E1 128.543} C_DIS
LIN {X -0.003,Y -293.401,Z 832.714,A 0.000,B 0.000,C 90.000,E1 128.508} C_DIS
LIN {X -0.062,Y -298.727,Z 832.713,A 0.000,B 0.000,C 90.000,E1 128.338} C_DIS
LIN {X -0.117,Y -301.043,Z 832.712,A 0.000,B 0.000,C 90.000,E1 128.177} C_DIS
LIN {X 0.012,Y -304.190,Z 832.710,A 0.000,B 0.000,C 90.000,E1 127.810} C_DIS
LIN {X -0.071,Y -306.183,Z 832.708,A 0.000,B 0.000,C 90.000,E1 127.523} C_DIS
LIN {X -0.154,Y -307.745,Z 832.707,A 0.000,B 0.000,C 90.000,E1 127.237} C_DIS
LIN {X 0.058,Y -309.084,Z 832.705,A 0.000,B 0.000,C 90.000,E1 126.870} C_DIS
LIN {X 0.144,Y -320.179,Z 832.685,A 0.000,B 0.000,C 90.000,E1 123.293} C_DIS
LIN {X -0.017,Y -330.533,Z 832.669,A 0.000,B 0.000,C 90.000,E1 120.463} C_DIS
LIN {X 0.067,Y -342.239,Z 832.654,A 0.000,B 0.000,C 90.000,E1 117.641} C_DIS
LIN {X 0.019,Y -355.391,Z 832.638,A 0.000,B 0.000,C 90.000,E1 114.899} C_DIS
LIN {X -0.037,Y -368.396,Z 832.625,A 0.000,B 0.000,C 90.000,E1 112.514} C_DIS
LIN {X -0.056,Y -382.733,Z 832.612,A 0.000,B 0.000,C 90.000,E1 110.174} C_DIS
LIN {X 0.020,Y -398.504,Z 832.599,A 0.000,B 0.000,C 90.000,E1 107.873} C_DIS
LIN {X -0.135,Y -415.824,Z 832.587,A 0.000,B 0.000,C 90.000,E1 105.662} C_DIS
LIN {X -0.073,Y -434.806,Z 832.575,A 0.000,B 0.000,C 90.000,E1 103.480} C_DIS
LIN {X 0.038,Y -454.882,Z 832.563,A 0.000,B 0.000,C 90.000,E1 101.422} C_DIS
LIN {X -0.148,Y -467.691,Z 832.557,A 0.000,B 0.000,C 90.000,E1 100.254} C_DIS
LIN {X -0.141,Y -469.745,Z 832.556,A 0.000,B 0.000,C 90.000,E1 100.018} C_DIS
LIN {X -0.135,Y -471.306,Z 832.554,A 0.000,B 0.000,C 90.000,E1 99.782} C_DIS
LIN {X 0.105,Y -472.586,Z 832.553,A 0.000,B 0.000,C 90.000,E1 99.500} C_DIS
LIN {X -0.041,Y -473.528,Z 832.551,A 0.000,B 0.000,C 90.000,E1 99.265} C_DIS
LIN {X 0.073,Y -474.571,Z 832.549,A 0.000,B 0.000,C 90.000,E1 98.746} C_DIS
LIN {X -0.206,Y -474.627,Z 832.546,A 0.000,B 0.000,C 90.000,E1 98.276} C_DIS
LIN {X -0.078,Y -473.708,Z 832.543,A 0.000,B 0.000,C 90.000,E1 97.757} C_DIS
LIN {X 0.050,Y -471.663,Z 832.540,A 0.000,B 0.000,C 90.000,E1 97.239} C_DIS
LIN {X -0.104,Y -461.813,Z 832.532,A 0.000,B 0.000,C 90.000,E1 95.739} C_DIS
LIN {X 0.171,Y -444.888,Z 832.516,A 0.000,B 0.000,C 90.000,E1 92.865} C_DIS
LIN {X -0.056,Y -435.669,Z 832.507,A 0.000,B 0.000,C 90.000,E1 91.318} C_DIS
LIN {X -0.012,Y -426.120,Z 832.498,A 0.000,B 0.000,C 90.000,E1 89.714} C_DIS
LIN {X -0.021,Y -414.685,Z 832.488,A 0.000,B 0.000,C 90.000,E1 87.822} C_DIS
LIN {X 0.076,Y -404.814,Z 832.479,A 0.000,B 0.000,C 90.000,E1 86.159} C_DIS
LIN {X 0.137,Y -391.650,Z 832.466,A 0.000,B 0.000,C 90.000,E1 83.913} C_DIS
LIN {X -0.059,Y -378.776,Z 832.454,A 0.000,B 0.000,C 90.000,E1 81.659} C_DIS
LIN {X -0.165,Y -363.149,Z 832.437,A 0.000,B 0.000,C 90.000,E1 78.757} C_DIS
LIN {X -0.001,Y -352.692,Z 832.426,A 0.000,B 0.000,C 90.000,E1 76.645} C_DIS
LIN {X 0.019,Y -342.275,Z 832.414,A 0.000,B 0.000,C 90.000,E1 74.519} C_DIS
LIN {X -0.023,Y -330.442,Z 832.400,A 0.000,B 0.000,C 90.000,E1 72.054} C_DIS
LIN {X 0.114,Y -320.278,Z 832.388,A 0.000,B 0.000,C 90.000,E1 69.826} C_DIS
LIN {X 0.091,Y -306.237,Z 832.370,A 0.000,B 0.000,C 90.000,E1 66.613} C_DIS
LIN {X 0.146,Y -294.218,Z 832.354,A 0.000,B 0.000,C 90.000,E1 63.640} C_DIS
LIN {X 0.037,Y -283.954,Z 832.339,A 0.000,B 0.000,C 90.000,E1 60.973} C_DIS
LIN {X 0.076,Y -271.597,Z 832.320,A 0.000,B 0.000,C 90.000,E1 57.533} C_DIS
LIN {X -0.045,Y -261.152,Z 832.302,A 0.000,B 0.000,C 90.000,E1 54.402} C_DIS
LIN {X 0.013,Y -251.170,Z 832.284,A 0.000,B 0.000,C 90.000,E1 51.170} C_DIS
LIN {X -0.100,Y -240.746,Z 832.264,A 0.000,B 0.000,C 90.000,E1 47.553} C_DIS
LIN {X 0.099,Y -231.130,Z 832.243,A 0.000,B 0.000,C 90.000,E1 43.785} C_DIS
LIN {X -0.002,Y -223.896,Z 832.227,A 0.000,B 0.000,C 90.000,E1 40.782} C_DIS
LIN {X -0.086,Y -216.884,Z 832.209,A 0.000,B 0.000,C 90.000,E1 37.729} C_DIS
LIN {X 0.054,Y -208.783,Z 832.188,A 0.000,B 0.000,C 90.000,E1 33.785} C_DIS
LIN {X 0.127,Y -202.777,Z 832.170,A 0.000,B 0.000,C 90.000,E1 30.590} C_DIS
LIN {X 0.090,Y -197.435,Z 832.152,A 0.000,B 0.000,C 90.000,E1 27.385} C_DIS
LIN {X 0.013,Y -192.799,Z 832.134,A 0.000,B 0.000,C 90.000,E1 24.155} C_DIS
LIN {X 0.027,Y -189.009,Z 832.116,A 0.000,B 0.000,C 90.000,E1 20.865} C_DIS
LIN {X -0.015,Y -185.298,Z 832.093,A 0.000,B 0.000,C 90.000,E1 16.732} C_DIS
LIN {X -0.010,Y -182.353,Z 832.065,A 0.000,B 0.000,C 90.000,E1 11.715} C_DIS
LIN {X -0.021,Y -183.248,Z 831.969,A 0.000,B 0.000,C 90.000,E1 354.489} C_DIS
LIN {X 0.021,Y -186.613,Z 831.941,A 0.000,B 0.000,C 90.000,E1 349.454} C_DIS
LIN {X 0.083,Y -190.411,Z 831.918,A 0.000,B 0.000,C 90.000,E1 345.283} C_DIS
LIN {X -0.100,Y -195.113,Z 831.896,A 0.000,B 0.000,C 90.000,E1 341.221} C_DIS
LIN {X 0.060,Y -200.690,Z 831.873,A 0.000,B 0.000,C 90.000,E1 337.102} C_DIS
LIN {X -0.103,Y -207.049,Z 831.851,A 0.000,B 0.000,C 90.000,E1 333.127} C_DIS
LIN {X 0.041,Y -214.336,Z 831.829,A 0.000,B 0.000,C 90.000,E1 329.125} C_DIS
LIN {X 0.024,Y -222.411,Z 831.807,A 0.000,B 0.000,C 90.000,E1 325.229} C_DIS
LIN {X -0.112,Y -229.555,Z 831.790,A 0.000,B 0.000,C 90.000,E1 322.190} C_DIS
LIN {X -0.031,Y -238.437,Z 831.771,A 0.000,B 0.000,C 90.000,E1 318.771} C_DIS
LIN {X 0.110,Y -248.098,Z 831.752,A 0.000,B 0.000,C 90.000,E1 315.405} C_DIS
LIN {X 0.011,Y -258.740,Z 831.734,A 0.000,B 0.000,C 90.000,E1 312.162} C_DIS
LIN {X 0.051,Y -270.206,Z 831.716,A 0.000,B 0.000,C 90.000,E1 308.955} C_DIS
LIN {X -0.055,Y -282.570,Z 831.699,A 0.000,B 0.000,C 90.000,E1 305.851} C_DIS
LIN {X -0.081,Y -297.688,Z 831.680,A 0.000,B 0.000,C 90.000,E1 302.467} C_DIS
LIN {X 0.118,Y -312.806,Z 831.664,A 0.000,B 0.000,C 90.000,E1 299.461} C_DIS
LIN {X -0.153,Y -325.765,Z 831.651,A 0.000,B 0.000,C 90.000,E1 297.257} C_DIS
LIN {X 0.126,Y -343.930,Z 831.636,A 0.000,B 0.000,C 90.000,E1 294.387} C_DIS
LIN {X -0.087,Y -356.971,Z 831.625,A 0.000,B 0.000,C 90.000,E1 292.589} C_DIS
LIN {X -0.025,Y -370.946,Z 831.615,A 0.000,B 0.000,C 90.000,E1 290.791} C_DIS
LIN {X 0.241,Y -396.310,Z 831.599,A 0.000,B 0.000,C 90.000,E1 287.873} C_DIS
LIN {X -0.039,Y -411.757,Z 831.590,A 0.000,B 0.000,C 90.000,E1 286.260} C_DIS
LIN {X 0.038,Y -424.394,Z 831.583,A 0.000,B 0.000,C 90.000,E1 284.898} C_DIS
LIN {X -0.224,Y -436.729,Z 831.575,A 0.000,B 0.000,C 90.000,E1 283.592} C_DIS
LIN {X 0.169,Y -446.219,Z 831.569,A 0.000,B 0.000,C 90.000,E1 282.479} C_DIS
LIN {X -0.198,Y -455.173,Z 831.564,A 0.000,B 0.000,C 90.000,E1 281.478} C_DIS
LIN {X -0.025,Y -463.520,Z 831.558,A 0.000,B 0.000,C 90.000,E1 280.423} C_DIS
LIN {X -0.139,Y -469.414,Z 831.554,A 0.000,B 0.000,C 90.000,E1 279.670} C_DIS
LIN {X 0.122,Y -476.416,Z 831.548,A 0.000,B 0.000,C 90.000,E1 278.624} C_DIS
LIN {X 0.117,Y -480.925,Z 831.544,A 0.000,B 0.000,C 90.000,E1 277.871} C_DIS
LIN {X 0.094,Y -484.747,Z 831.540,A 0.000,B 0.000,C 90.000,E1 277.125} C_DIS
LIN {X 0.163,Y -487.906,Z 831.536,A 0.000,B 0.000,C 90.000,E1 276.372} C_DIS
LIN {X -0.124,Y -489.578,Z 831.533,A 0.000,B 0.000,C 90.000,E1 275.910} C_DIS
LIN {X 0.085,Y -490.878,Z 831.530,A 0.000,B 0.000,C 90.000,E1 275.391} C_DIS
LIN {X -0.229,Y -491.831,Z 831.527,A 0.000,B 0.000,C 90.000,E1 274.935} C_DIS
LIN {X -0.001,Y -492.477,Z 831.525,A 0.000,B 0.000,C 90.000,E1 274.416} C_DIS
LIN {X 0.230,Y -492.706,Z 831.522,A 0.000,B 0.000,C 90.000,E1 273.898} C_DIS
LIN {X -0.060,Y -492.581,Z 831.519,A 0.000,B 0.000,C 90.000,E1 273.440} C_DIS
LIN {X 0.173,Y -492.057,Z 831.516,A 0.000,B 0.000,C 90.000,E1 272.922} C_DIS
LIN {X -0.113,Y -491.162,Z 831.514,A 0.000,B 0.000,C 90.000,E1 272.465} C_DIS
LIN {X 0.094,Y -489.751,Z 831.511,A 0.000,B 0.000,C 90.000,E1 271.949} C_DIS
LIN {X -0.180,Y -487.971,Z 831.508,A 0.000,B 0.000,C 90.000,E1 271.489} C_DIS
LIN {X 0.012,Y -485.599,Z 831.505,A 0.000,B 0.000,C 90.000,E1 270.974} C_DIS
LIN {X 0.187,Y -482.650,Z 831.503,A 0.000,B 0.000,C 90.000,E1 270.458} C_DIS
LIN {X -0.135,Y -479.045,Z 831.500,A 0.000,B 0.000,C 90.000,E1 270.000} C_DIS
LIN {X 0.006,Y -474.620,Z 831.497,A 0.000,B 0.000,C 90.000,E1 269.484} C_DIS
LIN {X -0.172,Y -472.110,Z 831.496,A 0.000,B 0.000,C 90.000,E1 269.255} C_DIS
LIN {X 0.119,Y -466.407,Z 831.493,A 0.000,B 0.000,C 90.000,E1 268.740} C_DIS
LIN {X 0.117,Y -463.301,Z 831.492,A 0.000,B 0.000,C 90.000,E1 268.511} C_DIS
LIN {X 0.094,Y -456.623,Z 831.490,A 0.000,B 0.000,C 90.000,E1 268.108} C_DIS
LIN {X 0.182,Y -449.374,Z 831.488,A 0.000,B 0.000,C 90.000,E1 267.764} C_DIS
LIN {X -0.056,Y -441.851,Z 831.486,A 0.000,B 0.000,C 90.000,E1 267.535} C_DIS
LIN {X 0.149,Y -433.213,Z 831.485,A 0.000,B 0.000,C 90.000,E1 267.306} C_DIS
LIN {X 0.003,Y -423.483,Z 831.484,A 0.000,B 0.000,C 90.000,E1 267.192} C_DIS
LIN {X 0.187,Y -417.586,Z 831.484,A 0.000,B 0.000,C 90.000,E1 267.135} C_DIS
LIN {X 0.047,Y -181.008,Z 831.484,A 0.000,B 0.000,C 90.000,E1 267.135} C_DIS
LIN {X 0.030,Y -180.906,Z 831.475,A 0.000,B 0.000,C 90.000,E1 265.412} C_DIS
LIN {X -0.094,Y -180.714,Z 831.470,A 0.000,B 0.000,C 90.000,E1 264.609} C_DIS
LIN {X 0.004,Y -178.801,Z 831.442,A 0.000,B 0.000,C 90.000,E1 259.511} C_DIS
LIN {X 0.081,Y -175.847,Z 831.413,A 0.000,B 0.000,C 90.000,E1 254.393} C_DIS
LIN {X 0.041,Y -172.582,Z 831.390,A 0.000,B 0.000,C 90.000,E1 250.134} C_DIS
LIN {X 0.057,Y -171.470,Z 831.380,A 0.000,B 0.000,C 90.000,E1 248.411} C_DIS
